(* CoDeSys 2.3.9.50 project: Acp_Bag_2Wrapping_Code.pro *)
(* Libraries: COMlibV2.lib 24.2.14 07:15:46, SysLibAlarmTrend.lib 17.10.05 06:42:38, TcBase.lib 14.5.09 05:44:08, TcSystem.lib 7.6.16 04:31:22, TcUtilities.lib 3.2.16 09:38:58, STANDARD.LIB 5.6.98 05:33:02, TcEtherCAT.lib 30.11.16 13:22:18, SysLibTargetVisu.lib 16.6.08 09:54:26, TcBaseMath.lib 27.7.04 05:37:56, SysLibVisu.lib 7.7.04 11:47:22, TcSystemCX.lib 7.9.16 06:21:26, FB_DateTime.lib 15.2.16 11:06:26, TcMath.lib 23.9.04 08:45:30 *)

(* Task configuration *)
TASK Standard (PRIORITY := 0, INTERVAL := T#10ms);
	MAIN
END_TASK
TASK VISU_TASK (PRIORITY := 3, INTERVAL := T#200ms);
	MAINTARGETVISU_PAINT_CODE
END_TASK
TASK VISU_INPUT_TASK (PRIORITY := 2, INTERVAL := T#50ms);
	MAINTARGETVISU_INPUT_CODE
END_TASK

(* Global variable list: Alarms *)
VAR_GLOBAL
	bAError1: BOOL;
	bAError2: BOOL;
	bAError3: BOOL;
	bAError4: BOOL;
	bAError5: BOOL;
	bAError6: BOOL;
	bAError7: BOOL;
	bAError8: BOOL;
	bAError9: BOOL;
	bAError10: BOOL;
	bAError11: BOOL;
	bAError12: BOOL;
	bAError13: BOOL;
	bAError14: BOOL;
	bAError15: BOOL;
	bAError16: BOOL;
	bAError17: BOOL;
	bAError18: BOOL;
	bAError19: BOOL;
	bAError20: BOOL;
	bAError1Status: STRING;
	bAError2Status: STRING;
	bAError3Status: STRING;
	bAError4Status: STRING;
	bAError5Status: STRING;
	bAError6Status: STRING;
	bAError7Status: STRING;
	bAError8Status: STRING;
	bAError9Status: STRING;
	bAError10Status: STRING;
	bAError11Status: STRING;
	bAError12Status: STRING;
	bAError13Status: STRING;
	bAError14Status: STRING;
	bAError15Status: STRING;
	bAError16Status: STRING;
	bAError17Status: STRING;
	bAError18Status: STRING;
	bAError19Status: STRING;
	bAError20Status: STRING;
END_VAR

(* Global variable list: Auto *)
VAR_GLOBAL
	bQAFeedingConveyorMotor: BOOL;
	bAConeFeedConveyorStart: BOOL;
	bAConeFeedConWait: BOOL;
	bRConePresentInConeFeedCon: BOOL;

	bAConeFeedingPistonHomeRsError: BOOL;
	bQAConeFeedPisOn: BOOL;

	bASealConRdy: BOOL;
	bQAForwardPistonOn: BOOL;
	bQAReversePistonOn: BOOL;

	bAConeTiltingRdy: BOOL;
	ConeFeedPistonRdy: BOOL;
	bAConeFeedCount: BOOL;
	bAConeFeedPisOn: BOOL;
	bAConeFeedingPistonEndRsError: BOOL;
	Cone1Reached: BOOL;
	bAConeFeededCount: INT;
	Cone2Reached: BOOL;
	TotalNoOfCones: INT;

	bAConeFwdRevRdy: BOOL;
	bATiltingPistonOn: BOOL;
	bAConeTiltingPistonEndRsError: BOOL;
	bAFwdRevPisRdy: BOOL;
	bAFwdRevCom: BOOL;
	bAConeTiltingPistonHomeRsError: BOOL;
	bATiltingCylCom: BOOL;
	bAConeTiltingCount: INT;

	bAWrapRdy: BOOL;
	bAForwardPistonOn: BOOL;
	bAReversePistonOn: BOOL;
	bAForwardPisEndRsError: BOOL;
	bAReversePisEndRsError: BOOL;
	bAFwdRevCount: INT;
	bAForwardPisHomeRsError: BOOL;
	bAReversePisHomeRsError: BOOL;
	bAWrappingConRdy: BOOL;

	bAWrapConRdy: BOOL;
	bAWrappingConOn: BOOL;
	bAWrapConeAlaignError: BOOL;
	bAWrapConeAlaignError1: BOOL;
	bAWrappingPisRdy: BOOL;
	bAWrapPiston1On: BOOL;
	bAWrapPiston2On: BOOL;
	bASealingConRdy: BOOL;
	bASheetFeedError: BOOL;
	bAWrapPis1EndRsError: BOOL;
	bAWrapPis2EndRsError: BOOL;
	bAWrappingPisCylCom: BOOL;
	bAWrappingPisCylComInt: BOOL;
	bASealUnitStart: BOOL;


	iBagRowCounter_243: INT;
	bQAColumnStopperPiston: BOOL;
	bABagOperationStarted_243: BOOL;
	bABagUnitRdy_243: BOOL;
	bABagOperationRdy_243: BOOL;
	bQAConePusher2Piston: BOOL;
	bQAColumnReversePiston: BOOL;
	bQAConePusher1Piston: BOOL;
	bABagHalfOpCom_243: BOOL;
	bABagOperationStarted: BOOL;
	bABagOperationComplete: BOOL;
	bQABagHolder: BOOL;
	bQASeparatorplatePiston: BOOL;
	bQABagUp_Down50piston: BOOL;
	bABagOperationComplete_243: BOOL;
	bQABagPusherForwardPiston: BOOL;
	bQABagPusherReversePiston: BOOL;
	TON_bagPusher_243: TON;
	BagOpCom_243: BOOL;
	bForceBagHolder: BOOL;
	bABagComplete: BOOL;
	bQABagTiltingpistonReverse: BOOL;
	bABagTiltingRevOk_243: BOOL;
	bQAColumnConeReversePiston: BOOL;
	bQABagUp_Down180piston: BOOL;
	bQABagTiltingpistonForward: BOOL;
	bQABagBagUp_Down50piston: BOOL;
	bQABagRowHolderpiston: BOOL;

	bASealingConRdy_Bag: BOOL;
	bASealingConRdy_Box: BOOL;
	bASealingUnitOperationCom: BOOL;
	bABoxUnitRdy: BOOL;
	bABoxOperationCom: BOOL;
	bQASealingConFwd1: BOOL;
	bQASealingConRev: BOOL;
	bASealConeSet1Started: BOOL;
	bQASealingConFwd2: BOOL;
	bASealingConeCountEnable: BOOL;
	bASealConeSet1Completed: BOOL;
	bASealConeSet2Started: BOOL;
	bASealConeSet2Completed: BOOL;
	bASealConeRevSetCompleted: BOOL;
	bASealConeMissError: BOOL;
	bASealConeMissErrorStatus: STRING;
	bASealConeMissError1: BOOL;
	bASealConeMissError2: BOOL;
	bASealConeMissError3: BOOL;
	bASealingUnitInt: BOOL;
	bQASealingSeparatorYAxisPiston: BOOL;
	bQASealingTopPiston: BOOL;
	bQASealingBottomPiston: BOOL;
	bQASealingSeparatorXAxisPiston: BOOL;
	bAFilmLoaded1: BOOL;
	bAFilmLoaded2: BOOL;
END_VAR

(* Global variable list: DataLog *)
VAR_GLOBAL
	R_TRIG_IndoPrint: R_TRIG;
	FB_FileOpen_Indo: FB_FileOpen;
	FB_FileWrite_Indo: FB_FileWrite;
	FB_FileClose_Indo: FB_FileClose;
	FB_FileDelete_Indo: FB_FileDelete;
	IndoReport: INT;
	ReportHead1_Indo: BOOL;
	ST1_ProductionData: BOOL;
	ReportHead2_Indo: BOOL;
	ReportBot1_Indo: BOOL;
	stStation1_ProductionData: BOOL;
	ReportBot2_Indo: BOOL;
	testbit: BOOL;
	sOldDay: STRING;
	WriteError: INT;
	OpenError: INT;
	ProductionData_IndoPrint2:STRING(255);
	ProductionDataError_IndoPrint2:STRING(255);
	ProductionDataValues_IndoPrint_Com:STRING(255);
	bANewDay: BOOL;
	SerialNoError: DINT;
	ProductionDataValues_IndoPrint: STRING(255);
	ProductionData_IndoPrint: STRING(255);
	ProductionDataError_IndoPrint: STRING(255);
	ProductionData_ReportData1 : ProductionData_ReportData;
	PROCESSCOMPLETE: BOOL;
	ReportSave: BOOL;
	SerialNo AT %Q*: DINT;
END_VAR

(* Global variable list: Initialize *)
VAR_GLOBAL
	Initialize_TapHmi: BOOL;
	bAInitializeSeq: BOOL;
	bAMachineOn: BOOL;
	bASupplyPressureError: BOOL;
	IntAllOver: BOOL;
	bAIntHomeCheckError: BOOL;

	bQRWappingConveyorMotor: BOOL;
	WrappingConIntRunning: BOOL;
	WrapConIntOver: BOOL;
	bRConePresentInWrapCon: BOOL;
	bQRWrappingPiston1: BOOL;
	bQRWrappingPiston2: BOOL;
	bAWrappingPiston1RsError: BOOL;
	bAWrappingPiston2RsError: BOOL;
	WrapUnitIntOver: BOOL;
	sWrappingConStatus: STRING;
	TiltIntRdy: BOOL;

	bQRForwardPiston: BOOL;
	bQRReversePiston: BOOL;
	bQRTiltingPiston: BOOL;
	bQATiltingPiston: BOOL;
	TiltingIntOvr: BOOL;

	bQRSealingConveyorMotor: BOOL;
	bRConePresentInSealCon: BOOL;
	SealingConIntRunning: BOOL;
	sSealingConStatus: STRING;
	SealConIntOver: BOOL;
	bQRSealingTopPiston: BOOL;
	bQRSealingBottomPiston: BOOL;
	bQRSealingSeparatorXAxisPiston: BOOL;
	bRSealUnitIntOver: BOOL;
	bQRSealingSeparatorYAxisPiston: BOOL;

	bRBagUnitIntRdy: BOOL;
END_VAR

(* Global variable list: Inputs *)
VAR_GLOBAL
					(*I1-EL1809*)

	(*IR1*)	bIUnit_A_RowStopperHome AT %I* : BOOL;
	(*IR2*)	bIUnit_A_RowStopperMiddle AT %I* :BOOL;
	(*IR3*)	bIUnit_A_RowStopperEnd AT %I* :BOOL;
	(*IR4*)	bIUnit_B_RowStopperHome AT %I* :BOOL;
	(*IR5*)	bIUnit_B_RowStopperMiddle AT %I* :BOOL;
	(*IR6*)	bIUnit_B_RowStopperEnd AT %I* :BOOL;
	(*IR7*)	bIUnit_A_ConeDetectionSensor1 AT %I* :BOOL;
	(*IR8*)	bIUnit_A_ConeDetectionSensor2 AT %I* :BOOL;
	(*IR9*)	bIUnit_A_ConeDetectionSensor3 AT %I* :BOOL;
	(*IR10*)	bIUnit_A_ConeDetectionSensor4 AT %I* :BOOL;
	(*IR11*)	bIUnit_A_ConeCrossLimitSwitch AT %I* :BOOL;
	(*IR12*)	bIUnit_B_ConeDetectionSensor1 AT %I* :BOOL;
	(*IR13*)	bIUnit_B_ConeDetectionSensor2 AT %I* :BOOL;
	(*IR14*)	bIUnit_B_ConeDetectionSensor3 AT %I* :BOOL;
	(*IR15*)	bIUnit_B_ConeDetectionSensor4 AT %I* :BOOL;
	(*IR16*)	bIUnit_B_ConeCrossLimitSwitch AT %I* :BOOL;


					(*I2-EL1809*)

	(*IR17*)	bIUnit_AStartPb AT %I* :BOOL;
	(*IR18*)	bIUnit_BStartPb AT %I* :BOOL;
	(*IR19*)	bISpare1 AT %I* :BOOL;
	(*IW1*)	bIMcStartPb AT %I* :BOOL;
	(*IW2*)	bIMcStopPb AT %I* :BOOL;
	(*IW3*)	bIAutoManualSwitch AT %I* :BOOL;
	(*IW4*)	bIEmergencySwitchPb AT %I* :BOOL;
	(*IW5*)	bIProgramKeySwitch AT %I* :BOOL;
	(*IW6*)	bIConeOrientationTopLimitSwitch AT %I* :BOOL;
	(*IW7*)	bIFeedconeStopSensor AT %I* :BOOL;
	(*IW8*)	bIConeFeedingPistonHome AT%I* :BOOL;
	(*IW9*)	bIConeFeedingPistonEnd AT %I* :BOOL;
	(*IW10*)	bIForwardPistonHome AT %I* :BOOL;
	(*IW11*)	bIForwardPistonEnd AT %I* :BOOL;
	(*IW12*)	bIReversePistonHome AT %I* :BOOL;
	(*IW13*)	bIReversePistonEnd AT %I* :BOOL;

						(*I3-EL1809*)

	(*IW14*)	bITiltingHome AT %I* :BOOL;
	(*IW15*)	bITiltingMiddle AT %I* :BOOL;
	(*IW16*)	bITiltingEnd AT %I* :BOOL;
	(*IW17*)	bIWrappingChanelPiston1Home AT %I* :BOOL;
	(*IW18*)	bIWrappingChanelPiston1Middle AT %I* :BOOL;
	(*IW19*)	bIWrappingChanelPiston1End AT %I* :BOOL;
	(*IW20*)	bIWrappingChanelPiston2Home AT %I* :BOOL;
	(*IW21*)	bIWrappingChanelPiston2Middle AT %I* :BOOL;
	(*IW22*)	bIWrappingChanelPiston2End AT %I* :BOOL;
	(*IW23*)	bIWrappingCone1 AT %I* :BOOL;
	(*IW24*)	bIWrappingCone2 AT %I* :BOOL;
	(*IW25*)	bIFilmTensionRod1Home AT %I* :BOOL;
	(*IW26*)	bIFilmTensionRod1End AT %I* :BOOL;
	(*IW27*)	bIFilmTensionRod2Home AT %I* :BOOL;
	(*IW28*)	bIFilmTensionRod2End AT %I* :BOOL;
	(*IW29*)	bISpare2 AT %I* :BOOL;

						(*I4-EL1809*)

	(*IW30*)	bISealingSeparatorYAxisPistonHome AT %I* :BOOL;
	(*IW31*)	bISealingSeparatorYAxisPistoEnd AT %I* :BOOL;
	(*IW32*)	bISealingTopPistonHome AT %I* :BOOL;
	(*IW33*)	bISealingTopPistonEnd AT %I* :BOOL;
	(*IW34*)	bISealingBottomPistonHome AT %I* :BOOL;
	(*IW35*)	bISealingBottomPistonEnd AT %I* :BOOL;
	(*IW36*)	bISealingSeparatorXAxisPistonHome AT %I* :BOOL;
	(*IW37*)	bISealingSeparatorXAxisPistonEnd AT %I* :BOOL;
	(*IW38*)	bIManualSealingPb AT %I* :BOOL;
	(*IW39*)	bIConeCountsensor AT %I* :BOOL;
	(*IW40*)	bIPressureSwitch AT %I* :BOOL;
	(*IW41*)	bIResetPb AT %I* :BOOL;
	(*IW42*)	bIPausePb AT %I* :BOOL;
	(*IW43*)	bIConeCountSensorRev AT %I* :BOOL;
	(*IW44*)	bIConecountStopperPistonHome AT %I* :BOOL;
	(*IW45*)	bIConecountStopperPistonEnd AT%I* :BOOL;


						(*I5-EL1809*)

	(*IW46*)	bIResetSealingPb AT %I* :BOOL;
	(*IW47*)	bISpare4 AT %I* :BOOL;
	(*IW48*)	bISpare5 AT %I* :BOOL;
	(*IW49*)	bISpare6 AT %I* :BOOL;
	(*IW50*)	bISpare7 AT %I* :BOOL;
	(*IW51*)	bISpare8 AT %I* :BOOL;
	(*IW52*)	bISpare9 AT %I* :BOOL;
	(*IW53*)	bISpare10 AT %I*: BOOL;

					(*I6-EL1809*)

	(*IB1*)	bIColumnStopperPistonHome AT %I*: BOOL;
	(*IB2*)	bIColumnStopperPistonEnd AT %I*: BOOL;
	(*IB3*)	bIColumnReversePistonHome AT %I*: BOOL;
	(*IB4*)	bIColumnReversePistonEnd AT %I*: BOOL;
	(*IB5*)	bISeperatorPlatePistonHome AT %I*: BOOL;
	(*IB6*)	bISeperatorPlatePistonEnd AT %I*: BOOL;
	(*IB7*)	bIConePusher1PistonHome AT %I*: BOOL;
	(*IB8*)	bIConePusher1PistonEnd AT %I*: BOOL;
	(*IB9*)	bIConePusher1SaftyObjectSensor AT %I*: BOOL;
	(*IB10*)	bIBagUpDown180PistonHome AT %I*: BOOL;
	(*IB11*)	bIBagUpDown180PistonEnd AT %I*: BOOL;
	(*IB12*)	bIBagUpDown50PistonHome AT %I*: BOOL;
	(*IB13*)	bIBagUpDown50PistonEnd AT %I*: BOOL;
	(*IB14*)	bIBagPusherPistonHome AT %I*: BOOL;
	(*IB15*)	bIBagPusherPistonMiddle AT %I*: BOOL;
	(*IB16*)	bIBagPusherPistonEnd AT %I*: BOOL;

						(*I7-EL1809*)

	(*IB17*)	bIBagTiltingPistonHome AT %I*: BOOL;
	(*IB18*)	bIBagiltingPistonEnd AT %I*: BOOL;
	(*IB19*)	bIBagEmptyCheckObjectSensor AT %I*: BOOL;
	(*IB20*)	bIBagHolderOn  AT %I*: BOOL;
	(*IB21*)	bIBagResetPb AT %I*: BOOL;
	(*IB22*) 	bISpare11 AT %I*: BOOL;
	(*IB23*) 	bISpare12 AT %I*: BOOL;
	(*IB24*) 	bISpare13 AT %I*: BOOL;
END_VAR

(* Global variable list: Main *)
VAR_GLOBAL
	(****************START / STOP / PAUSE / RESUME***************)
	Start_TapHmi: BOOL;
	bAutoModeOn: BOOL;
	bMcStartInAuto: BOOL;
	bMcStopEnable: BOOL;
	Stop_TapHmi: BOOL;
	Pause_TapHmi: BOOL;
	bPauseSeq: BOOL;
	Resume_TapHmi: BOOL;
	Reset_TapHmi: BOOL;
	bErrorReset: BOOL;
	bMcStopEnable1: BOOL;
(*============== Auto/Manual Mode Selection Logic========================*)
	bManualModeOn: BOOL;
	bManualmode: BOOL;
	sMcStatus: STRING;
	bHidePopUp: BOOL;
	bManualModeOk_TapHmi: BOOL;
	bManualModeNOk_TapHmi: BOOL;
(*====================Logic for Model Selection===============*)
	BagSelect_TapHmi: BOOL;
	bAMainIntStarted: BOOL;
	bABoxModeSelected: BOOL;
	BoxSelect_TapHmi: BOOL;
	bABagModeSelected: BOOL;
	sPackingModeStatus: STRING;

	(****************DATE AND TIME***********)
	FB_DateTime_1: FB_DateTime;
	sHourPreFix: STRING;
	sHou: STRING;
	sDayPreFix: STRING;
	sDay: STRING;
	sMonthPreFix: STRING;
	sMonth: STRING;
	sDayF: STRING;
	sMonthF: STRING;
	sDayMonth: STRING;
	sDayF1: STRING;
	sMonthF1: STRING;
	sDayMonth1: STRING;
	sDayMonthYear: STRING;
	sDayMonthYear1: STRING;
	sDaateReport: STRING;
	ReportPath: STRING;
	ReportPath_Final: STRING;
	ReportPath_Final_1: STRING;
	ReportPath_Final_2: STRING;
	sDateReport: STRING;
	ReportPathError: STRING;
	ReportPath_FinalError: STRING;
	ReportPath_Final_1Error: STRING;
	ReportPath_Final_2Error: STRING;
	DateTimeVar: STRING;
	wTodayToHmiFinal: STRING;
(*===============Shift Calculation============*)
	bAShift1Hour: BOOL;
	bAShift2Hour: BOOL;
	bAShift3Hour: BOOL;
	Sfiht1From_Hmi  AT %Q*: WORD;
	Sfiht2From_Hmi  AT %Q*: WORD;
	Sfiht3From_Hmi  AT %Q*: WORD;
	Sfiht1To_Hmi AT %Q*: WORD;
	Sfiht2To_Hmi AT %Q*: WORD;
	Sfiht3To_Hmi AT %Q*: WORD;
	sShitStatus: STRING;
END_VAR

(* Global variable list: Manual *)
VAR_GLOBAL
	WrappingSafety: BOOL;
	SealingSafety: BOOL;
	bManualSealEnable: BOOL;
	bManualSealEnable2: BOOL;
	bMManualSealOn: BOOL;
	bQM_Cone_Sealing_Bottom_Piston: BOOL;
	bQM_Cone_Sealing_Top_Piston: BOOL;
	bHMI_Cone_Forward_Piston_On: BOOL;
	bQM_Cone_Forward_Piston: BOOL;
	bHMI_Cone_Feeding_Piston_On: BOOL;
	bQM_Cone_Feeding_Piston: BOOL;
	bHMI_Cone_Reverse_Piston_On: BOOL;
	bQM_Cone_Reverse_Piston: BOOL;
	bHMI_Cone_Tilting_Piston_On: BOOL;
	bQM_Cone_Tilting_Piston: BOOL;
	bQM_Cone_Tilting_Piston_Rev: BOOL;
	bHMI_Cone_Tilting_Piston_On_Rev: BOOL;
	bHMI_Cone_Wrapping_Piston_On: BOOL;
	bQM_Cone_Wrapping_Piston_Rev: BOOL;
	bQM_Cone_Wrapping_Piston_Fwd: BOOL;
	bHMI_Cone_Wrapping_Piston_On_Rev: BOOL;
	bHMI_Cone_Sealing_Top_Piston_On: BOOL;
	bHMI_Cone_Sealing_Bottom_Piston_On: BOOL;
	bHMI_Cone_Sealing_YAxis_Piston_On: BOOL;
	bQM_Cone_Sealing_YAxis_Piston: BOOL;
	bHMI_Cone_Sealing_XAxis_Piston_On: BOOL;
	bQM_Cone_Sealing_XAxis_Piston: BOOL;
	bHMI_Cone_Feeding_Conveyor_On: BOOL;
	bQM_Cone_Feeding_Conveyor: BOOL;
	bHMI_Cone_Wrapping_Conveyor_On: BOOL;
	bQM_Cone_Wrapping_Conveyor: BOOL;
	bHMI_Cone_Sealing_Conveyor_On: BOOL;
	bQM_Cone_Sealing_Conveyor: BOOL;
	bIConePusher1_On_Hmi: BOOL;
	bQMConePusher1: BOOL;
	bIConePusher2_On_Hmi: BOOL;
	bQMConePusher2: BOOL;
	bIConePusher3_On_Hmi: BOOL;
	bQMConePusher3: BOOL;
	bIBagPusherFwd_On_Hmi: BOOL;
	bQMBagPusherFwd: BOOL;
	bIBagPusherRev_On_Hmi: BOOL;
	bQMBagPusherRev: BOOL;
	bIUpDownPiston_1_On_Hmi: BOOL;
	bQMUpDownPiston_1: BOOL;
	bIUpDownPiston_2_On_Hmi: BOOL;
	bQMUpDownPiston_2: BOOL;
	bIBagTiltingFwd_On_Hmi: BOOL;
	bQMBagTiltingFwd: BOOL;
	bIBagTiltingRev_On_Hmi: BOOL;
	bQMBagTiltingRev: BOOL;
	bIColumn_Stopper_Piston_On_Hmi: BOOL;
	bQMColumnStopperPiston: BOOL;
	bIColumnConeForwardPiston_On_Hmi: BOOL;
	bQMColumnConeForwardPiston: BOOL;
	bIBagHolder_On: BOOL;
	bIBagHolder_On_Hmi: BOOL;
	bIBagPusherHome: BOOL;
	bQMBagHolderPiston: BOOL;
	bHMI_RetA_Fwd_On: BOOL;
	bHMI_RetA_Rev_On: BOOL;
	bQM_RetA_Rev: BOOL;
	bQM_RetA_Fwd: BOOL;
	bHMI_Ret_RevA_On: BOOL;

	bHMI_RetB_Fwd_On: BOOL;
	bHMI_RetB_Rev_On: BOOL;
	bQM_RetB_Rev: BOOL;
	bQM_RetB_Fwd: BOOL;
	bHMI_Ret_RevB_On: BOOL;
	bHMI_Cone_Wrapping_Piston1_On: BOOL;
	bQM_Cone_Wrapping_Piston1_Fwd: BOOL;
	bHMI_Cone_Wrapping_Piston1_On_Rev: BOOL;
	bQM_Cone_Wrapping_Piston1_Rev: BOOL;
	bHMI_Cone_Wrapping_Piston2_On: BOOL;
	bQM_Cone_Wrapping_Piston2_Rev: BOOL;
	bQM_Cone_Wrapping_Piston2_Fwd: BOOL;
	bHMI_Cone_Wrapping_Piston2_On_Rev: BOOL;
	bHMI_Cone_Count_Piston_On: BOOL;
	bQM_Cone_Count_Piston: BOOL;
	bIBagRowHolderPiston_On_Hmi: BOOL;
	bQMBagRowHolderPiston: BOOL;
END_VAR

(* Global variable list: Output_Flags *)
VAR_GLOBAL
	bQAFilmRollerMotor1OnAuto:BOOL;
	bQAFilmRollerMotor2OnAuto: BOOL;
	bQRColumnStopperPiston: BOOL;
	bQMColumnReversePiston: BOOL;
	bQMSeparatorplatePiston: BOOL;
	bQMConePusher1Piston: BOOL;
	bQMConePusher2Piston: BOOL;
	bQMBagPusherForwardPiston: BOOL;
	bQMBagPusherReversePiston: BOOL;
	bQMBagUp_Down180piston: BOOL;
	bQMBagUp_Down50piston: BOOL;
	bQMBagTiltingpistonForward: BOOL;
	bQMBagTiltingpistonReverse: BOOL;
	bQMSpareOutput13: BOOL;
	bQMSpareOutput14: BOOL;
	bQMSpareOutput15: BOOL;
	bQRColumnReversePiston: BOOL;
	bQRSeparatorplatePiston: BOOL;
	bQRConePusher1Piston: BOOL;
	bQRConePusher2Piston: BOOL;
	bQRBagPusherForwardPiston: BOOL;
	bQRBagPusherReversePiston: BOOL;
	bQRBagHolderpiston: BOOL;
	bQRBagUp_Down180piston: BOOL;
	bQRBagUp_Down50piston: BOOL;
	bQRBagTiltingpistonForward: BOOL;
	bQRBagTiltingpistonReverse: BOOL;
	bQRSpareOutput13: BOOL;
	bQRSpareOutput14: BOOL;
	bQRSpareOutput15: BOOL;
	bAQColumnReversePiston: BOOL;
	bQABagHolderpiston: BOOL;
	bQASpareOutput13: BOOL;
	bQASpareOutput14: BOOL;
	bQASpareOutput15: BOOL;
	bQMSpareOutput5: BOOL;
	bQRSpareOutput5: BOOL;
	bQASpareOutput5: BOOL;
	bQMSpareOutput6: BOOL;
	bQRSpareOutput6: BOOL;
	bQASpareOutput6: BOOL;
	bQMSpareOutput7: BOOL;
	bQRSpareOutput7: BOOL;
	bQASpareOutput7: BOOL;
	bQMSpareOutput8: BOOL;
	bQRSpareOutput8: BOOL;
	bQASpareOutput8: BOOL;
	bQMSpareOutput9: BOOL;
	bQRSpareOutput9: BOOL;
	bQASpareOutput9: BOOL;
	bQMSpareOutput10: BOOL;
	bQRSpareOutput10: BOOL;
	bQASpareOutput10: BOOL;
	bQMSpareOutput11: BOOL;
	bQRSpareOutput11: BOOL;
	bQASpareOutput11: BOOL;
	bQMSpareOutput12: BOOL;
	bQRSpareOutput12: BOOL;
	bQASpareOutput12: BOOL;
	bQMConeFeedingPiston: BOOL;
	bQRConeFeedingPiston: BOOL;
	bQMForwardPiston: BOOL;
	bQMReversePiston: BOOL;
	bQMTiltingPiston: BOOL;
	bQMWrappingPiston1: BOOL;
	bQMWrappingPiston2: BOOL;
	bQMSealingSeparatorYAxisPiston: BOOL;
	bQMSealingTopPiston: BOOL;
	bQMSealingBottomPiston: BOOL;
	bQMSealingSeparatorXAxisPiston: BOOL;
	bQMFilmRollerMotor1: BOOL;
	bQAFilmRollerMotor1: BOOL;
	bQMFilmRollerMotor2: BOOL;
	bQAFilmRollerMotor2: BOOL;
	bQMConeCountPiston: BOOL;
	bQAConeCountPiston: BOOL;
	bQMFeedingConveyorMotor: BOOL;
	bQMWappingConveyorMotor: BOOL;
	bQAWappingConveyorMotor: BOOL;
	bQMSealingConveyorMotor: BOOL;
	bQASealingConveyorMotor: BOOL;
	bQMRetA_RowStopperMotorFwd: BOOL;
	bQRRetA_RowStopperMotorFwd: BOOL;
	bQMRetA_RowStopperMotorRev: BOOL;
	bQRRetA_RowStopperMotorRev: BOOL;
	bQMRetB_RowStopperMotorFwd: BOOL;
	bQRRetB_RowStopperMotorFwd: BOOL;
	bQMRetB_RowStopperMotorRev: BOOL;
	bQRRetB_RowStopperMotorRev: BOOL;
	bQMSpareOutput1: BOOL;
	bQRSpareOutput1: BOOL;
	bQARetA_WeightOk: BOOL;
	bQARetA_WeightNOk: BOOL;
	bQARetB_WeightOk: BOOL;
	bQARetB_WeightNOk: BOOL;
	bQMSpareOutput2: BOOL;
	bQRSpareOutput2: BOOL;
	bQMSpareOutput3: BOOL;
	bQRSpareOutput3: BOOL;
	bQMSpareOutput4: BOOL;
	bQRSpareOutput4: BOOL;
	bQMTowerLampRed: BOOL;
	bQRTowerLampRed: BOOL;
	bQMTowerLampGreen: BOOL;
	bQRTowerLampGreen: BOOL;
	bQMTowerLampYellow: BOOL;
	bQRTowerLampYellow: BOOL;
	bQMTowerBuzzer: BOOL;
	bQRTowerBuzzer: BOOL;
	bQARetA_RowStopperMotorFwd: BOOL;
	bQARetA_RowStopperMotorRev: BOOL;
	bQARetB_RowStopperMotorFwd: BOOL;
	bQARetB_RowStopperMotorRev: BOOL;
	bQASpareOutput1: BOOL;
	bQASpareOutput2: BOOL;
	bQASpareOutput3: BOOL;
	bQASpareOutput4: BOOL;
	bQATowerLampRed: BOOL;
	bQATowerLampGreen: BOOL;
	bQATowerLampYellow: BOOL;
	bQATowerBuzzer: BOOL;
	bQAForwardPiston: BOOL;
	bQAReversePiston: BOOL;
	bQAWrappingPiston1: BOOL;
	bQAWrappingPiston2: BOOL;
	bQRConeCountPiston: BOOL;
	bQRFeedingConveyorMotor: BOOL;

	bQBagHolder: BOOL;
	bQAConePusher3Piston: BOOL;
	bAConePusher1SafetyError: BOOL;
	bAConePusher1SafetyErrorStatus: STRING;

END_VAR

(* Global variable list: Outputs *)
VAR_GLOBAL
				(*O1-EL2809*)

	bQRetA_RowStopperMotorFwd AT %Q* :BOOL;(*OR1*)
	bQRetA_RowStopperMotorRev AT %Q* :BOOL;(*OR2*)
	bQRetB_RowStopperMotorFwd AT %Q* :BOOL;(*OR3*)
	bQRetB_RowStopperMotorRev AT %Q* :BOOL;(*OR4*)
	bQSpareOutput1 AT %Q* :BOOL;(*OR5*)
	bQRetA_WeightOk AT %Q* :BOOL;(*OR6*)
	bQRetA_WeightNOk AT %Q* :BOOL;(*OR7*)
	bQRetB_WeightOk AT %Q* :BOOL;(*OR8*)
	bQRetB_WeightNOk AT %Q* :BOOL;(*OR9*)
	bQSpareOutput2 AT %Q* :BOOL;(*OR10*)
	bQSpareOutput3 AT %Q* :BOOL;(*OR11*)
	bQSpareOutput4 AT %Q* :BOOL;(*OR12*)
	bQTowerLampRed AT %Q* :BOOL;(*R1*)
	bQTowerLampGreen AT %Q* :BOOL;(*R2*)
	bQTowerLampYellow AT %Q* :BOOL;(*R3*)
	bQTowerBuzzer AT %Q* :BOOL;(*R4*)


			(*O2-EL2809*)

	bQConeFeedingPiston AT %Q* :BOOL;(*OW1*)
	bQForwardPiston AT %Q* :BOOL;(*OW2*)
	bQReversePiston AT %Q* :BOOL;(*OW3*)
	bQTiltingPiston AT %Q* :BOOL;(*OW4*)
	bQWrappingPiston1 AT %Q* :BOOL;(*OW5*)
	bQWrappingPiston2 AT %Q* :BOOL;(*OW6*)
	bQSealingSeparatorYAxisPiston AT %Q* :BOOL;(*OW7*)
	bQSealingTopPiston AT %Q* :BOOL;(*OW8*)
	bQSealingBottomPiston AT %Q* :BOOL;(*OW9*)
	bQSealingSeparatorXAxisPiston AT %Q* :BOOL;(*OW10*)
	bQFilmRollerMotor1 AT %Q* :BOOL;(*OW11*)
	bQFilmRollerMotor2 AT %Q* :BOOL;(*OW12*)
	bQConeCountPiston AT %Q* :BOOL;(*OW13*)
	bQFeedingConveyorMotor AT %Q* :BOOL;(*OW14*)
	bQWappingConveyorMotor AT %Q* :BOOL;(*OW15*)
	bQSealingConveyorMotor AT %Q* :BOOL;(*OW16*)



			(*O3-EL2008*)

	bQSpareOutput5 AT %Q* :BOOL;(*OW20*)
	bQSpareOutput6 AT %Q* :BOOL;(*OW21*)
	bQSpareOutput7 AT %Q* :BOOL;(*OW22*)
	bQSpareOutput8 AT %Q* :BOOL;(*OW23*)
	bQSpareOutput9 AT %Q* :BOOL;(*OW24*)
	bQSpareOutput10 AT %Q* :BOOL;(*OW25*)
	bQSpareOutput11 AT %Q* :BOOL;(*OW26*)
	bQSpareOutput12 AT %Q* :BOOL;(*OW27*)

			(*O4-EL2809*)

	bQColumnStopperPiston AT %Q* :BOOL;(*OB1*)
	bQColumnReversePiston AT %Q* :BOOL;(*OB2*)
	bQSeparatorplatePiston AT %Q* :BOOL;(*OB3*)
	bQConePusher1Piston AT %Q* :BOOL;(*OB4*)
	bQConePusher2Piston AT %Q* :BOOL;(*OB5*)
	bQBagPusherForwardPiston AT %Q* :BOOL;(*OB6*)
	bQBagPusherReversePiston AT %Q* :BOOL;(*OB7*)
	bQBagHolderpiston AT %Q* :BOOL;(*OB8*)
	bQBagUp_Down180piston AT %Q* :BOOL;(*OB9*)
	bQBagUp_Down50piston AT %Q* :BOOL;(*OB10*)
	bQBagTiltingpistonForward AT %Q* :BOOL;(*OB11*)
	bQBagTiltingpistonReverse AT %Q* :BOOL;(*OB12*)
	bQBagRowHolderpiston AT %Q* :BOOL;(*OB13*)
	bQSpareOutput13 AT %Q* :BOOL;(*OB14*)
	bQSpareOutput14 AT %Q* :BOOL;(*OB15*)
	bQSpareOutput15 AT %Q* :BOOL;(*OB16*)

END_VAR

(* Global variable list: Parameters *)
VAR_GLOBAL
	Default_NetWeight_Report: STRING;
	Default_GrossWeight_Report: STRING;
	Actual_NetWeight_Report: STRING;
	Actual_GrossWeight_Report: STRING;
	COUNT_DIS: STRING;
	BLEND_DIS: STRING;
	LOTNO_DIS: STRING;
	CARTONNO_DIS: DINT;
	SHADE_DIS: STRING;
END_VAR

(* Global variable list: Print *)
VAR_GLOBAL
	PrintEnabled: BOOL;
	PrintValue: INT;
	PrintEnable_TogHmi: BOOL;
	ProductionData_PrintData: ProductionData_PrintData;
	ProductionDataValues_Print: STRING(255);
	ProductionDataValues_Print_Com:STRING(255);
	ProductionData_Print: STRING(255);
	FB_FileOpen1: FB_FileOpen;
	FB_FileWrite1: FB_FileWrite;
	FB_FileClose1: FB_FileClose;
	FB_FileDelete1: FB_FileDelete;
	PrintOk: BOOL;
END_VAR

(* Global variable list: TwinCAT_Configuration *)
(* Generated automatically by TwinCAT - (read only) *)
VAR_CONFIG
	Weight_Read.COMin_1_COMPort_1 AT %IB0 : EL6inData22B;
	Weight_Read.COMOut_1_COMPort_1 AT %QB0 : EL6outData22B;
	Weight_Read.COMin_2_COMPort_2 AT %IB24 : EL6inData22B;
	Weight_Read.COMOut_2_COMPort_2 AT %QB24 : EL6outData22B;
	.SerialNo AT %QB48 : DINT;
	.bIUnit_A_RowStopperHome AT %IX48.0 : BOOL;	(*  ~ {LinkedWith:TIID^Device 3 (EtherCAT)^Term 1 (EK1100)^Term 2 (EL1809)^Channel 1^Input} *)
	.bIUnit_A_RowStopperMiddle AT %IX48.1 : BOOL;	(*  ~ {LinkedWith:TIID^Device 3 (EtherCAT)^Term 1 (EK1100)^Term 2 (EL1809)^Channel 2^Input} *)
	.bIUnit_A_RowStopperEnd AT %IX48.2 : BOOL;	(*  ~ {LinkedWith:TIID^Device 3 (EtherCAT)^Term 1 (EK1100)^Term 2 (EL1809)^Channel 3^Input} *)
	.bIUnit_B_RowStopperHome AT %IX48.3 : BOOL;	(*  ~ {LinkedWith:TIID^Device 3 (EtherCAT)^Term 1 (EK1100)^Term 2 (EL1809)^Channel 4^Input} *)
	.bIUnit_B_RowStopperMiddle AT %IX48.4 : BOOL;	(*  ~ {LinkedWith:TIID^Device 3 (EtherCAT)^Term 1 (EK1100)^Term 2 (EL1809)^Channel 5^Input} *)
	.bIUnit_B_RowStopperEnd AT %IX48.5 : BOOL;	(*  ~ {LinkedWith:TIID^Device 3 (EtherCAT)^Term 1 (EK1100)^Term 2 (EL1809)^Channel 6^Input} *)
	.bIUnit_A_ConeDetectionSensor1 AT %IX48.6 : BOOL;	(*  ~ {LinkedWith:TIID^Device 3 (EtherCAT)^Term 1 (EK1100)^Term 2 (EL1809)^Channel 7^Input} *)
	.bIUnit_A_ConeDetectionSensor2 AT %IX48.7 : BOOL;	(*  ~ {LinkedWith:TIID^Device 3 (EtherCAT)^Term 1 (EK1100)^Term 2 (EL1809)^Channel 8^Input} *)
	.bIUnit_A_ConeDetectionSensor3 AT %IX49.0 : BOOL;	(*  ~ {LinkedWith:TIID^Device 3 (EtherCAT)^Term 1 (EK1100)^Term 2 (EL1809)^Channel 9^Input} *)
	.bIUnit_A_ConeDetectionSensor4 AT %IX49.1 : BOOL;	(*  ~ {LinkedWith:TIID^Device 3 (EtherCAT)^Term 1 (EK1100)^Term 2 (EL1809)^Channel 10^Input} *)
	.bIUnit_A_ConeCrossLimitSwitch AT %IX49.2 : BOOL;	(*  ~ {LinkedWith:TIID^Device 3 (EtherCAT)^Term 1 (EK1100)^Term 2 (EL1809)^Channel 11^Input} *)
	.bIUnit_B_ConeDetectionSensor1 AT %IX49.3 : BOOL;	(*  ~ {LinkedWith:TIID^Device 3 (EtherCAT)^Term 1 (EK1100)^Term 2 (EL1809)^Channel 12^Input} *)
	.bIUnit_B_ConeDetectionSensor2 AT %IX49.4 : BOOL;	(*  ~ {LinkedWith:TIID^Device 3 (EtherCAT)^Term 1 (EK1100)^Term 2 (EL1809)^Channel 13^Input} *)
	.bIUnit_B_ConeDetectionSensor3 AT %IX49.5 : BOOL;	(*  ~ {LinkedWith:TIID^Device 3 (EtherCAT)^Term 1 (EK1100)^Term 2 (EL1809)^Channel 14^Input} *)
	.bIUnit_B_ConeDetectionSensor4 AT %IX49.6 : BOOL;	(*  ~ {LinkedWith:TIID^Device 3 (EtherCAT)^Term 1 (EK1100)^Term 2 (EL1809)^Channel 15^Input} *)
	.bIUnit_B_ConeCrossLimitSwitch AT %IX49.7 : BOOL;	(*  ~ {LinkedWith:TIID^Device 3 (EtherCAT)^Term 1 (EK1100)^Term 2 (EL1809)^Channel 16^Input} *)
	.bIUnit_AStartPb AT %IX50.0 : BOOL;	(*  ~ {LinkedWith:TIID^Device 3 (EtherCAT)^Term 1 (EK1100)^Term 3 (EL1809)^Channel 1^Input} *)
	.bIUnit_BStartPb AT %IX50.1 : BOOL;	(*  ~ {LinkedWith:TIID^Device 3 (EtherCAT)^Term 1 (EK1100)^Term 3 (EL1809)^Channel 2^Input} *)
	.bISpare1 AT %IX50.2 : BOOL;	(*  ~ {LinkedWith:TIID^Device 3 (EtherCAT)^Term 1 (EK1100)^Term 3 (EL1809)^Channel 3^Input} *)
	.bIMcStartPb AT %IX50.3 : BOOL;	(*  ~ {LinkedWith:TIID^Device 3 (EtherCAT)^Term 1 (EK1100)^Term 3 (EL1809)^Channel 4^Input} *)
	.bIMcStopPb AT %IX50.4 : BOOL;	(*  ~ {LinkedWith:TIID^Device 3 (EtherCAT)^Term 1 (EK1100)^Term 3 (EL1809)^Channel 5^Input} *)
	.bIAutoManualSwitch AT %IX50.5 : BOOL;	(*  ~ {LinkedWith:TIID^Device 3 (EtherCAT)^Term 1 (EK1100)^Term 3 (EL1809)^Channel 6^Input} *)
	.bIEmergencySwitchPb AT %IX50.6 : BOOL;	(*  ~ {LinkedWith:TIID^Device 3 (EtherCAT)^Term 1 (EK1100)^Term 3 (EL1809)^Channel 7^Input} *)
	.bIProgramKeySwitch AT %IX50.7 : BOOL;	(*  ~ {LinkedWith:TIID^Device 3 (EtherCAT)^Term 1 (EK1100)^Term 3 (EL1809)^Channel 8^Input} *)
	.bIConeOrientationTopLimitSwitch AT %IX51.0 : BOOL;	(*  ~ {LinkedWith:TIID^Device 3 (EtherCAT)^Term 1 (EK1100)^Term 3 (EL1809)^Channel 9^Input} *)
	.bIFeedconeStopSensor AT %IX51.1 : BOOL;	(*  ~ {LinkedWith:TIID^Device 3 (EtherCAT)^Term 1 (EK1100)^Term 3 (EL1809)^Channel 10^Input} *)
	.bIConeFeedingPistonHome AT %IX51.2 : BOOL;	(*  ~ {LinkedWith:TIID^Device 3 (EtherCAT)^Term 1 (EK1100)^Term 3 (EL1809)^Channel 11^Input} *)
	.bIConeFeedingPistonEnd AT %IX51.3 : BOOL;	(*  ~ {LinkedWith:TIID^Device 3 (EtherCAT)^Term 1 (EK1100)^Term 3 (EL1809)^Channel 12^Input} *)
	.bIForwardPistonHome AT %IX51.4 : BOOL;	(*  ~ {LinkedWith:TIID^Device 3 (EtherCAT)^Term 1 (EK1100)^Term 3 (EL1809)^Channel 13^Input} *)
	.bIForwardPistonEnd AT %IX51.5 : BOOL;	(*  ~ {LinkedWith:TIID^Device 3 (EtherCAT)^Term 1 (EK1100)^Term 3 (EL1809)^Channel 14^Input} *)
	.bIReversePistonHome AT %IX51.6 : BOOL;	(*  ~ {LinkedWith:TIID^Device 3 (EtherCAT)^Term 1 (EK1100)^Term 3 (EL1809)^Channel 15^Input} *)
	.bIReversePistonEnd AT %IX51.7 : BOOL;	(*  ~ {LinkedWith:TIID^Device 3 (EtherCAT)^Term 1 (EK1100)^Term 3 (EL1809)^Channel 16^Input} *)
	.bITiltingHome AT %IX52.0 : BOOL;	(*  ~ {LinkedWith:TIID^Device 3 (EtherCAT)^Term 1 (EK1100)^Term 4 (EL1809)^Channel 1^Input} *)
	.bITiltingMiddle AT %IX52.1 : BOOL;	(*  ~ {LinkedWith:TIID^Device 3 (EtherCAT)^Term 1 (EK1100)^Term 4 (EL1809)^Channel 2^Input} *)
	.bITiltingEnd AT %IX52.2 : BOOL;	(*  ~ {LinkedWith:TIID^Device 3 (EtherCAT)^Term 1 (EK1100)^Term 4 (EL1809)^Channel 3^Input} *)
	.bIWrappingChanelPiston1Home AT %IX52.3 : BOOL;	(*  ~ {LinkedWith:TIID^Device 3 (EtherCAT)^Term 1 (EK1100)^Term 4 (EL1809)^Channel 4^Input} *)
	.bIWrappingChanelPiston1Middle AT %IX52.4 : BOOL;	(*  ~ {LinkedWith:TIID^Device 3 (EtherCAT)^Term 1 (EK1100)^Term 4 (EL1809)^Channel 5^Input} *)
	.bIWrappingChanelPiston1End AT %IX52.5 : BOOL;	(*  ~ {LinkedWith:TIID^Device 3 (EtherCAT)^Term 1 (EK1100)^Term 4 (EL1809)^Channel 6^Input} *)
	.bIWrappingChanelPiston2Home AT %IX52.6 : BOOL;	(*  ~ {LinkedWith:TIID^Device 3 (EtherCAT)^Term 1 (EK1100)^Term 4 (EL1809)^Channel 7^Input} *)
	.bIWrappingChanelPiston2Middle AT %IX52.7 : BOOL;	(*  ~ {LinkedWith:TIID^Device 3 (EtherCAT)^Term 1 (EK1100)^Term 4 (EL1809)^Channel 8^Input} *)
	.bIWrappingChanelPiston2End AT %IX53.0 : BOOL;	(*  ~ {LinkedWith:TIID^Device 3 (EtherCAT)^Term 1 (EK1100)^Term 4 (EL1809)^Channel 9^Input} *)
	.bIWrappingCone1 AT %IX53.1 : BOOL;	(*  ~ {LinkedWith:TIID^Device 3 (EtherCAT)^Term 1 (EK1100)^Term 4 (EL1809)^Channel 10^Input} *)
	.bIWrappingCone2 AT %IX53.2 : BOOL;	(*  ~ {LinkedWith:TIID^Device 3 (EtherCAT)^Term 1 (EK1100)^Term 4 (EL1809)^Channel 11^Input} *)
	.bIFilmTensionRod1Home AT %IX53.3 : BOOL;	(*  ~ {LinkedWith:TIID^Device 3 (EtherCAT)^Term 1 (EK1100)^Term 4 (EL1809)^Channel 12^Input} *)
	.bIFilmTensionRod1End AT %IX53.4 : BOOL;	(*  ~ {LinkedWith:TIID^Device 3 (EtherCAT)^Term 1 (EK1100)^Term 4 (EL1809)^Channel 13^Input} *)
	.bIFilmTensionRod2Home AT %IX53.5 : BOOL;	(*  ~ {LinkedWith:TIID^Device 3 (EtherCAT)^Term 1 (EK1100)^Term 4 (EL1809)^Channel 14^Input} *)
	.bIFilmTensionRod2End AT %IX53.6 : BOOL;	(*  ~ {LinkedWith:TIID^Device 3 (EtherCAT)^Term 1 (EK1100)^Term 4 (EL1809)^Channel 15^Input} *)
	.bISpare2 AT %IX53.7 : BOOL;	(*  ~ {LinkedWith:TIID^Device 3 (EtherCAT)^Term 1 (EK1100)^Term 4 (EL1809)^Channel 16^Input} *)
	.bISealingSeparatorYAxisPistonHome AT %IX54.0 : BOOL;	(*  ~ {LinkedWith:TIID^Device 3 (EtherCAT)^Term 1 (EK1100)^Term 5 (EL1809)^Channel 1^Input} *)
	.bISealingSeparatorYAxisPistoEnd AT %IX54.1 : BOOL;	(*  ~ {LinkedWith:TIID^Device 3 (EtherCAT)^Term 1 (EK1100)^Term 5 (EL1809)^Channel 2^Input} *)
	.bISealingTopPistonHome AT %IX54.2 : BOOL;	(*  ~ {LinkedWith:TIID^Device 3 (EtherCAT)^Term 1 (EK1100)^Term 5 (EL1809)^Channel 3^Input} *)
	.bISealingTopPistonEnd AT %IX54.3 : BOOL;	(*  ~ {LinkedWith:TIID^Device 3 (EtherCAT)^Term 1 (EK1100)^Term 5 (EL1809)^Channel 4^Input} *)
	.bISealingBottomPistonHome AT %IX54.4 : BOOL;	(*  ~ {LinkedWith:TIID^Device 3 (EtherCAT)^Term 1 (EK1100)^Term 5 (EL1809)^Channel 5^Input} *)
	.bISealingBottomPistonEnd AT %IX54.5 : BOOL;	(*  ~ {LinkedWith:TIID^Device 3 (EtherCAT)^Term 1 (EK1100)^Term 5 (EL1809)^Channel 6^Input} *)
	.bISealingSeparatorXAxisPistonHome AT %IX54.6 : BOOL;	(*  ~ {LinkedWith:TIID^Device 3 (EtherCAT)^Term 1 (EK1100)^Term 5 (EL1809)^Channel 7^Input} *)
	.bISealingSeparatorXAxisPistonEnd AT %IX54.7 : BOOL;	(*  ~ {LinkedWith:TIID^Device 3 (EtherCAT)^Term 1 (EK1100)^Term 5 (EL1809)^Channel 8^Input} *)
	.bIManualSealingPb AT %IX55.0 : BOOL;	(*  ~ {LinkedWith:TIID^Device 3 (EtherCAT)^Term 1 (EK1100)^Term 5 (EL1809)^Channel 9^Input} *)
	.bIConeCountsensor AT %IX55.1 : BOOL;	(*  ~ {LinkedWith:TIID^Device 3 (EtherCAT)^Term 1 (EK1100)^Term 5 (EL1809)^Channel 10^Input} *)
	.bIPressureSwitch AT %IX55.2 : BOOL;	(*  ~ {LinkedWith:TIID^Device 3 (EtherCAT)^Term 1 (EK1100)^Term 5 (EL1809)^Channel 11^Input} *)
	.bIResetPb AT %IX55.3 : BOOL;	(*  ~ {LinkedWith:TIID^Device 3 (EtherCAT)^Term 1 (EK1100)^Term 5 (EL1809)^Channel 12^Input} *)
	.bIPausePb AT %IX55.4 : BOOL;	(*  ~ {LinkedWith:TIID^Device 3 (EtherCAT)^Term 1 (EK1100)^Term 5 (EL1809)^Channel 13^Input} *)
	.bIConeCountSensorRev AT %IX55.5 : BOOL;	(*  ~ {LinkedWith:TIID^Device 3 (EtherCAT)^Term 1 (EK1100)^Term 5 (EL1809)^Channel 14^Input} *)
	.bIConecountStopperPistonHome AT %IX55.6 : BOOL;	(*  ~ {LinkedWith:TIID^Device 3 (EtherCAT)^Term 1 (EK1100)^Term 5 (EL1809)^Channel 15^Input} *)
	.bIConecountStopperPistonEnd AT %IX55.7 : BOOL;	(*  ~ {LinkedWith:TIID^Device 3 (EtherCAT)^Term 1 (EK1100)^Term 5 (EL1809)^Channel 16^Input} *)
	.bIResetSealingPb AT %IX56.0 : BOOL;	(*  ~ {LinkedWith:TIID^Device 3 (EtherCAT)^Term 1 (EK1100)^Term 7 (EL1008)^Channel 6^Input} *)
	.bISpare4 AT %IX56.1 : BOOL;	(*  ~ {LinkedWith:TIID^Device 3 (EtherCAT)^Term 1 (EK1100)^Term 8 (EL1008)^Channel 1^Input} *)
	.bISpare5 AT %IX56.2 : BOOL;	(*  ~ {LinkedWith:TIID^Device 3 (EtherCAT)^Term 1 (EK1100)^Term 8 (EL1008)^Channel 2^Input} *)
	.bISpare6 AT %IX56.3 : BOOL;	(*  ~ {LinkedWith:TIID^Device 3 (EtherCAT)^Term 1 (EK1100)^Term 8 (EL1008)^Channel 3^Input} *)
	.bISpare7 AT %IX56.4 : BOOL;	(*  ~ {LinkedWith:TIID^Device 3 (EtherCAT)^Term 1 (EK1100)^Term 8 (EL1008)^Channel 4^Input} *)
	.bISpare8 AT %IX56.5 : BOOL;	(*  ~ {LinkedWith:TIID^Device 3 (EtherCAT)^Term 1 (EK1100)^Term 8 (EL1008)^Channel 5^Input} *)
	.bISpare9 AT %IX56.6 : BOOL;	(*  ~ {LinkedWith:TIID^Device 3 (EtherCAT)^Term 1 (EK1100)^Term 8 (EL1008)^Channel 6^Input} *)
	.bISpare10 AT %IX56.7 : BOOL;	(*  ~ {LinkedWith:TIID^Device 3 (EtherCAT)^Term 1 (EK1100)^Term 8 (EL1008)^Channel 7^Input} *)
	.bIColumnStopperPistonHome AT %IX57.0 : BOOL;	(*  ~ {LinkedWith:TIID^Device 3 (EtherCAT)^Term 1 (EK1100)^Term 6 (EL1809)^Channel 1^Input} *)
	.bIColumnStopperPistonEnd AT %IX57.1 : BOOL;	(*  ~ {LinkedWith:TIID^Device 3 (EtherCAT)^Term 1 (EK1100)^Term 6 (EL1809)^Channel 2^Input} *)
	.bIColumnReversePistonHome AT %IX57.2 : BOOL;	(*  ~ {LinkedWith:TIID^Device 3 (EtherCAT)^Term 1 (EK1100)^Term 6 (EL1809)^Channel 3^Input} *)
	.bIColumnReversePistonEnd AT %IX57.3 : BOOL;	(*  ~ {LinkedWith:TIID^Device 3 (EtherCAT)^Term 1 (EK1100)^Term 6 (EL1809)^Channel 4^Input} *)
	.bISeperatorPlatePistonHome AT %IX57.4 : BOOL;	(*  ~ {LinkedWith:TIID^Device 3 (EtherCAT)^Term 1 (EK1100)^Term 6 (EL1809)^Channel 5^Input} *)
	.bISeperatorPlatePistonEnd AT %IX57.5 : BOOL;	(*  ~ {LinkedWith:TIID^Device 3 (EtherCAT)^Term 1 (EK1100)^Term 6 (EL1809)^Channel 6^Input} *)
	.bIConePusher1PistonHome AT %IX57.6 : BOOL;	(*  ~ {LinkedWith:TIID^Device 3 (EtherCAT)^Term 1 (EK1100)^Term 6 (EL1809)^Channel 7^Input} *)
	.bIConePusher1PistonEnd AT %IX57.7 : BOOL;	(*  ~ {LinkedWith:TIID^Device 3 (EtherCAT)^Term 1 (EK1100)^Term 6 (EL1809)^Channel 8^Input} *)
	.bIConePusher1SaftyObjectSensor AT %IX58.0 : BOOL;	(*  ~ {LinkedWith:TIID^Device 3 (EtherCAT)^Term 1 (EK1100)^Term 6 (EL1809)^Channel 9^Input} *)
	.bIBagUpDown180PistonHome AT %IX58.1 : BOOL;	(*  ~ {LinkedWith:TIID^Device 3 (EtherCAT)^Term 1 (EK1100)^Term 6 (EL1809)^Channel 10^Input} *)
	.bIBagUpDown180PistonEnd AT %IX58.2 : BOOL;	(*  ~ {LinkedWith:TIID^Device 3 (EtherCAT)^Term 1 (EK1100)^Term 6 (EL1809)^Channel 11^Input} *)
	.bIBagUpDown50PistonHome AT %IX58.3 : BOOL;	(*  ~ {LinkedWith:TIID^Device 3 (EtherCAT)^Term 1 (EK1100)^Term 6 (EL1809)^Channel 12^Input} *)
	.bIBagUpDown50PistonEnd AT %IX58.4 : BOOL;	(*  ~ {LinkedWith:TIID^Device 3 (EtherCAT)^Term 1 (EK1100)^Term 6 (EL1809)^Channel 13^Input} *)
	.bIBagPusherPistonHome AT %IX58.5 : BOOL;	(*  ~ {LinkedWith:TIID^Device 3 (EtherCAT)^Term 1 (EK1100)^Term 6 (EL1809)^Channel 14^Input} *)
	.bIBagPusherPistonMiddle AT %IX58.6 : BOOL;	(*  ~ {LinkedWith:TIID^Device 3 (EtherCAT)^Term 1 (EK1100)^Term 6 (EL1809)^Channel 15^Input} *)
	.bIBagPusherPistonEnd AT %IX58.7 : BOOL;	(*  ~ {LinkedWith:TIID^Device 3 (EtherCAT)^Term 1 (EK1100)^Term 6 (EL1809)^Channel 16^Input} *)
	.bIBagTiltingPistonHome AT %IX59.0 : BOOL;	(*  ~ {LinkedWith:TIID^Device 3 (EtherCAT)^Term 1 (EK1100)^Term 7 (EL1008)^Channel 1^Input} *)
	.bIBagiltingPistonEnd AT %IX59.1 : BOOL;	(*  ~ {LinkedWith:TIID^Device 3 (EtherCAT)^Term 1 (EK1100)^Term 7 (EL1008)^Channel 2^Input} *)
	.bIBagEmptyCheckObjectSensor AT %IX59.2 : BOOL;	(*  ~ {LinkedWith:TIID^Device 3 (EtherCAT)^Term 1 (EK1100)^Term 7 (EL1008)^Channel 3^Input} *)
	.bIBagHolderOn AT %IX59.3 : BOOL;	(*  ~ {LinkedWith:TIID^Device 3 (EtherCAT)^Term 1 (EK1100)^Term 7 (EL1008)^Channel 4^Input} *)
	.bIBagResetPb AT %IX59.4 : BOOL;	(*  ~ {LinkedWith:TIID^Device 3 (EtherCAT)^Term 1 (EK1100)^Term 7 (EL1008)^Channel 5^Input} *)
	.bISpare11 AT %IX59.5 : BOOL;	(*  ~ {LinkedWith:TIID^Device 3 (EtherCAT)^Term 1 (EK1100)^Term 8 (EL1008)^Channel 8^Input} *)
	.bISpare12 AT %IX59.6 : BOOL;	(*  ~ {LinkedWith:TIID^Device 3 (EtherCAT)^Term 1 (EK1100)^Term 7 (EL1008)^Channel 7^Input} *)
	.bISpare13 AT %IX59.7 : BOOL;	(*  ~ {LinkedWith:TIID^Device 3 (EtherCAT)^Term 1 (EK1100)^Term 7 (EL1008)^Channel 8^Input} *)
	.Sfiht1From_Hmi AT %QB52 : WORD;
	.Sfiht2From_Hmi AT %QB54 : WORD;
	.Sfiht3From_Hmi AT %QB56 : WORD;
	.Sfiht1To_Hmi AT %QB58 : WORD;
	.Sfiht2To_Hmi AT %QB60 : WORD;
	.Sfiht3To_Hmi AT %QB62 : WORD;
	.bQRetA_RowStopperMotorFwd AT %QX64.0 : BOOL;	(*  ~ {LinkedWith:TIID^Device 3 (EtherCAT)^Term 1 (EK1100)^Term 9 (EL2809)^Channel 1^Output} *)
	.bQRetA_RowStopperMotorRev AT %QX64.1 : BOOL;	(*  ~ {LinkedWith:TIID^Device 3 (EtherCAT)^Term 1 (EK1100)^Term 9 (EL2809)^Channel 2^Output} *)
	.bQRetB_RowStopperMotorFwd AT %QX64.2 : BOOL;	(*  ~ {LinkedWith:TIID^Device 3 (EtherCAT)^Term 1 (EK1100)^Term 9 (EL2809)^Channel 3^Output} *)
	.bQRetB_RowStopperMotorRev AT %QX64.3 : BOOL;	(*  ~ {LinkedWith:TIID^Device 3 (EtherCAT)^Term 1 (EK1100)^Term 9 (EL2809)^Channel 4^Output} *)
	.bQSpareOutput1 AT %QX64.4 : BOOL;	(*  ~ {LinkedWith:TIID^Device 3 (EtherCAT)^Term 1 (EK1100)^Term 9 (EL2809)^Channel 5^Output} *)
	.bQRetA_WeightOk AT %QX64.5 : BOOL;	(*  ~ {LinkedWith:TIID^Device 3 (EtherCAT)^Term 1 (EK1100)^Term 9 (EL2809)^Channel 6^Output} *)
	.bQRetA_WeightNOk AT %QX64.6 : BOOL;	(*  ~ {LinkedWith:TIID^Device 3 (EtherCAT)^Term 1 (EK1100)^Term 9 (EL2809)^Channel 7^Output} *)
	.bQRetB_WeightOk AT %QX64.7 : BOOL;	(*  ~ {LinkedWith:TIID^Device 3 (EtherCAT)^Term 1 (EK1100)^Term 9 (EL2809)^Channel 8^Output} *)
	.bQRetB_WeightNOk AT %QX65.0 : BOOL;	(*  ~ {LinkedWith:TIID^Device 3 (EtherCAT)^Term 1 (EK1100)^Term 9 (EL2809)^Channel 9^Output} *)
	.bQSpareOutput2 AT %QX65.1 : BOOL;	(*  ~ {LinkedWith:TIID^Device 3 (EtherCAT)^Term 1 (EK1100)^Term 9 (EL2809)^Channel 14^Output} *)
	.bQSpareOutput3 AT %QX65.2 : BOOL;	(*  ~ {LinkedWith:TIID^Device 3 (EtherCAT)^Term 1 (EK1100)^Term 9 (EL2809)^Channel 15^Output} *)
	.bQSpareOutput4 AT %QX65.3 : BOOL;	(*  ~ {LinkedWith:TIID^Device 3 (EtherCAT)^Term 1 (EK1100)^Term 9 (EL2809)^Channel 16^Output} *)
	.bQTowerLampRed AT %QX65.4 : BOOL;	(*  ~ {LinkedWith:TIID^Device 3 (EtherCAT)^Term 1 (EK1100)^Term 9 (EL2809)^Channel 10^Output} *)
	.bQTowerLampGreen AT %QX65.5 : BOOL;	(*  ~ {LinkedWith:TIID^Device 3 (EtherCAT)^Term 1 (EK1100)^Term 9 (EL2809)^Channel 11^Output} *)
	.bQTowerLampYellow AT %QX65.6 : BOOL;	(*  ~ {LinkedWith:TIID^Device 3 (EtherCAT)^Term 1 (EK1100)^Term 9 (EL2809)^Channel 12^Output} *)
	.bQTowerBuzzer AT %QX65.7 : BOOL;	(*  ~ {LinkedWith:TIID^Device 3 (EtherCAT)^Term 1 (EK1100)^Term 9 (EL2809)^Channel 13^Output} *)
	.bQConeFeedingPiston AT %QX66.0 : BOOL;	(*  ~ {LinkedWith:TIID^Device 3 (EtherCAT)^Term 1 (EK1100)^Term 10 (EL2809)^Channel 1^Output} *)
	.bQForwardPiston AT %QX66.1 : BOOL;	(*  ~ {LinkedWith:TIID^Device 3 (EtherCAT)^Term 1 (EK1100)^Term 10 (EL2809)^Channel 2^Output} *)
	.bQReversePiston AT %QX66.2 : BOOL;	(*  ~ {LinkedWith:TIID^Device 3 (EtherCAT)^Term 1 (EK1100)^Term 10 (EL2809)^Channel 3^Output} *)
	.bQTiltingPiston AT %QX66.3 : BOOL;	(*  ~ {LinkedWith:TIID^Device 3 (EtherCAT)^Term 1 (EK1100)^Term 10 (EL2809)^Channel 4^Output} *)
	.bQWrappingPiston1 AT %QX66.4 : BOOL;	(*  ~ {LinkedWith:TIID^Device 3 (EtherCAT)^Term 1 (EK1100)^Term 10 (EL2809)^Channel 5^Output} *)
	.bQWrappingPiston2 AT %QX66.5 : BOOL;	(*  ~ {LinkedWith:TIID^Device 3 (EtherCAT)^Term 1 (EK1100)^Term 10 (EL2809)^Channel 6^Output} *)
	.bQSealingSeparatorYAxisPiston AT %QX66.6 : BOOL;	(*  ~ {LinkedWith:TIID^Device 3 (EtherCAT)^Term 1 (EK1100)^Term 10 (EL2809)^Channel 7^Output} *)
	.bQSealingTopPiston AT %QX66.7 : BOOL;	(*  ~ {LinkedWith:TIID^Device 3 (EtherCAT)^Term 1 (EK1100)^Term 10 (EL2809)^Channel 8^Output} *)
	.bQSealingBottomPiston AT %QX67.0 : BOOL;	(*  ~ {LinkedWith:TIID^Device 3 (EtherCAT)^Term 1 (EK1100)^Term 10 (EL2809)^Channel 9^Output} *)
	.bQSealingSeparatorXAxisPiston AT %QX67.1 : BOOL;	(*  ~ {LinkedWith:TIID^Device 3 (EtherCAT)^Term 1 (EK1100)^Term 10 (EL2809)^Channel 10^Output} *)
	.bQFilmRollerMotor1 AT %QX67.2 : BOOL;	(*  ~ {LinkedWith:TIID^Device 3 (EtherCAT)^Term 1 (EK1100)^Term 10 (EL2809)^Channel 11^Output} *)
	.bQFilmRollerMotor2 AT %QX67.3 : BOOL;	(*  ~ {LinkedWith:TIID^Device 3 (EtherCAT)^Term 1 (EK1100)^Term 10 (EL2809)^Channel 12^Output} *)
	.bQConeCountPiston AT %QX67.4 : BOOL;	(*  ~ {LinkedWith:TIID^Device 3 (EtherCAT)^Term 1 (EK1100)^Term 10 (EL2809)^Channel 13^Output} *)
	.bQFeedingConveyorMotor AT %QX67.5 : BOOL;	(*  ~ {LinkedWith:TIID^Device 3 (EtherCAT)^Term 1 (EK1100)^Term 10 (EL2809)^Channel 14^Output} *)
	.bQWappingConveyorMotor AT %QX67.6 : BOOL;	(*  ~ {LinkedWith:TIID^Device 3 (EtherCAT)^Term 1 (EK1100)^Term 10 (EL2809)^Channel 15^Output} *)
	.bQSealingConveyorMotor AT %QX67.7 : BOOL;	(*  ~ {LinkedWith:TIID^Device 3 (EtherCAT)^Term 1 (EK1100)^Term 10 (EL2809)^Channel 16^Output} *)
	.bQSpareOutput5 AT %QX68.0 : BOOL;	(*  ~ {LinkedWith:TIID^Device 3 (EtherCAT)^Term 1 (EK1100)^Term 12 (EL2008)^Channel 1^Output} *)
	.bQSpareOutput6 AT %QX68.1 : BOOL;	(*  ~ {LinkedWith:TIID^Device 3 (EtherCAT)^Term 1 (EK1100)^Term 12 (EL2008)^Channel 2^Output} *)
	.bQSpareOutput7 AT %QX68.2 : BOOL;	(*  ~ {LinkedWith:TIID^Device 3 (EtherCAT)^Term 1 (EK1100)^Term 12 (EL2008)^Channel 3^Output} *)
	.bQSpareOutput8 AT %QX68.3 : BOOL;	(*  ~ {LinkedWith:TIID^Device 3 (EtherCAT)^Term 1 (EK1100)^Term 12 (EL2008)^Channel 4^Output} *)
	.bQSpareOutput9 AT %QX68.4 : BOOL;	(*  ~ {LinkedWith:TIID^Device 3 (EtherCAT)^Term 1 (EK1100)^Term 12 (EL2008)^Channel 5^Output} *)
	.bQSpareOutput10 AT %QX68.5 : BOOL;	(*  ~ {LinkedWith:TIID^Device 3 (EtherCAT)^Term 1 (EK1100)^Term 12 (EL2008)^Channel 6^Output} *)
	.bQSpareOutput11 AT %QX68.6 : BOOL;	(*  ~ {LinkedWith:TIID^Device 3 (EtherCAT)^Term 1 (EK1100)^Term 12 (EL2008)^Channel 7^Output} *)
	.bQSpareOutput12 AT %QX68.7 : BOOL;	(*  ~ {LinkedWith:TIID^Device 3 (EtherCAT)^Term 1 (EK1100)^Term 12 (EL2008)^Channel 8^Output} *)
	.bQColumnStopperPiston AT %QX69.0 : BOOL;	(*  ~ {LinkedWith:TIID^Device 3 (EtherCAT)^Term 1 (EK1100)^Term 11 (EL2809)^Channel 1^Output} *)
	.bQColumnReversePiston AT %QX69.1 : BOOL;	(*  ~ {LinkedWith:TIID^Device 3 (EtherCAT)^Term 1 (EK1100)^Term 11 (EL2809)^Channel 2^Output} *)
	.bQSeparatorplatePiston AT %QX69.2 : BOOL;	(*  ~ {LinkedWith:TIID^Device 3 (EtherCAT)^Term 1 (EK1100)^Term 11 (EL2809)^Channel 3^Output} *)
	.bQConePusher1Piston AT %QX69.3 : BOOL;	(*  ~ {LinkedWith:TIID^Device 3 (EtherCAT)^Term 1 (EK1100)^Term 11 (EL2809)^Channel 4^Output} *)
	.bQConePusher2Piston AT %QX69.4 : BOOL;	(*  ~ {LinkedWith:TIID^Device 3 (EtherCAT)^Term 1 (EK1100)^Term 11 (EL2809)^Channel 5^Output} *)
	.bQBagPusherForwardPiston AT %QX69.5 : BOOL;	(*  ~ {LinkedWith:TIID^Device 3 (EtherCAT)^Term 1 (EK1100)^Term 11 (EL2809)^Channel 6^Output} *)
	.bQBagPusherReversePiston AT %QX69.6 : BOOL;	(*  ~ {LinkedWith:TIID^Device 3 (EtherCAT)^Term 1 (EK1100)^Term 11 (EL2809)^Channel 7^Output} *)
	.bQBagHolderpiston AT %QX69.7 : BOOL;	(*  ~ {LinkedWith:TIID^Device 3 (EtherCAT)^Term 1 (EK1100)^Term 11 (EL2809)^Channel 8^Output} *)
	.bQBagUp_Down180piston AT %QX70.0 : BOOL;	(*  ~ {LinkedWith:TIID^Device 3 (EtherCAT)^Term 1 (EK1100)^Term 11 (EL2809)^Channel 9^Output} *)
	.bQBagUp_Down50piston AT %QX70.1 : BOOL;	(*  ~ {LinkedWith:TIID^Device 3 (EtherCAT)^Term 1 (EK1100)^Term 11 (EL2809)^Channel 10^Output} *)
	.bQBagTiltingpistonForward AT %QX70.2 : BOOL;	(*  ~ {LinkedWith:TIID^Device 3 (EtherCAT)^Term 1 (EK1100)^Term 11 (EL2809)^Channel 11^Output} *)
	.bQBagTiltingpistonReverse AT %QX70.3 : BOOL;	(*  ~ {LinkedWith:TIID^Device 3 (EtherCAT)^Term 1 (EK1100)^Term 11 (EL2809)^Channel 12^Output} *)
	.bQBagRowHolderpiston AT %QX70.4 : BOOL;	(*  ~ {LinkedWith:TIID^Device 3 (EtherCAT)^Term 1 (EK1100)^Term 11 (EL2809)^Channel 13^Output} *)
	.bQSpareOutput13 AT %QX70.5 : BOOL;	(*  ~ {LinkedWith:TIID^Device 3 (EtherCAT)^Term 1 (EK1100)^Term 11 (EL2809)^Channel 14^Output} *)
	.bQSpareOutput14 AT %QX70.6 : BOOL;	(*  ~ {LinkedWith:TIID^Device 3 (EtherCAT)^Term 1 (EK1100)^Term 11 (EL2809)^Channel 15^Output} *)
	.bQSpareOutput15 AT %QX70.7 : BOOL;	(*  ~ {LinkedWith:TIID^Device 3 (EtherCAT)^Term 1 (EK1100)^Term 11 (EL2809)^Channel 16^Output} *)
END_VAR

(* Data type *)
TYPE ProductionData_PrintData :
STRUCT
	Print:STRING;
	ConeType1:STRING;
	Blend1:STRING;
	DefaultnetWt1:STRING;
	DefaultGrossWt1:STRING;
	LotNo1:STRING;
	BagNo1:STRING;
	Shade1:STRING;
END_STRUCT
END_TYPE

(* Data type *)
TYPE ProductionData_ReportData :
STRUCT
	SERIALNO			:STRING;
	SDATE				:STRING;
	STIME				:STRING;
	BAGNO				:STRING;
	COUNTCODE		:STRING;
	LOTNO				:STRING;
	DFLTNETWEIGHT	:STRING;
	ACTNETWEIGHT		:STRING;
	DFLTGROSSWEIGHT	:STRING;
	ACTGROSSWEIGHT	:STRING;
END_STRUCT
END_TYPE

(* POU MAIN, ST *)
PROGRAM MAIN
	VAR

END_VAR
					(*START / STOP / PAUSE / RESUME*)


	IF (bIMcStartPb OR Start_TapHmi)  AND bAutoModeOn  THEN
	 bMcStartInAuto:=TRUE;
	bMcStopEnable:=FALSE;
	END_IF

	IF  bIMcStopPb OR Stop_TapHmi  OR NOT bAutoModeOn OR NOT bIEmergencySwitchPb THEN
	 bMcStartInAuto:=FALSE;bMcStopEnable:=TRUE;bMcStopEnable1:=TRUE;
	ELSE bMcStopEnable1:=FALSE;
	 END_IF

	IF Pause_TapHmi THEN
	bPauseSeq:=TRUE;END_IF
	IF Resume_TapHmi THEN
	bPauseSeq:=FALSE;END_IF

	IF bIResetPb OR Reset_TapHmi  OR bIResetSealingPb THEN
	bErrorReset:=TRUE;
	ELSE bErrorReset:=FALSE;END_IF

					(*============== Auto/Manual Mode Selection Logic========================*)

		IF bIAutoManualSwitch THEN
			bAutoModeOn:=TRUE; bManualModeOn:=FALSE;
		ELSIF  NOT bIAutoManualSwitch  THEN
			bManualModeOn:=TRUE; bAutoModeOn:=FALSE;
		END_IF

		IF bManualModeOn THEN sMcStatus:='Machine in Manual Mode';
		ELSIF bAutoModeOn THEN sMcStatus:='Machine in Auto Mode';
		END_IF

	IF bMcStartInAuto  AND NOT  bIAutoManualSwitch THEN
	bHidePopUp:=TRUE; END_IF

	IF NOT  bMcStartInAuto  AND NOT  bIAutoManualSwitch THEN
	bManualmode:=TRUE;  END_IF

	IF bHidePopUp AND bManualModeOk_TapHmi THEN
	bManualmode:=TRUE;bAutoModeOn:=FALSE;bHidePopUp:=FALSE; END_IF

	IF bHidePopUp AND bManualModeNOk_TapHmi THEN
	bHidePopUp:=FALSE; END_IF

					 (*====================Logic for Model Selection===============*)

		IF bAutoModeOn AND BagSelect_TapHmi AND NOT bAMainIntStarted THEN
		bABoxModeSelected:=FALSE;BoxSelect_TapHmi:=FALSE;bABagModeSelected:=TRUE; BoxSelect_TapHmi:=FALSE;
		ELSIF bAutoModeOn AND   BoxSelect_TapHmi AND NOT bAMainIntStarted THEN
		bABagModeSelected:=FALSE; BagSelect_TapHmi:=FALSE;bABoxModeSelected:=TRUE;
		END_IF

		IF bABagModeSelected THEN sPackingModeStatus:=' Bag Packing Selected '; END_IF
		IF bABoxModeSelected THEN sPackingModeStatus:=' Carton Packing Selected  '; END_IF




			(****************DATE AND TIME***********)

(*======================= RTC==============================*)

FB_DateTime_1(NET_ID:='5.69.70.240.1.1 ' , DATE_TIME=> );

IF FB_DateTime_1.FBLTIME.systemTime.wHour >0 AND  FB_DateTime_1.FBLTIME.systemTime.wHour<9 THEN
sHourPreFix:='0';sHou:=CONCAT(STR1:=sHourPreFix, Str2:=WORD_TO_STRING(FB_DateTime_1.FBLTIME.systemTime.wHour));
ELSIF FB_DateTime_1.FBLTIME.systemTime.wHour >=10 AND  FB_DateTime_1.FBLTIME.systemTime.wHour<=24 THEN
sHou:=WORD_TO_STRING(FB_DateTime_1.FBLTIME.systemTime.wHour);
END_IF

IF FB_DateTime_1.FBLTIME.systemTime.wDay >0 AND  FB_DateTime_1.FBLTIME.systemTime.wDay<10 THEN
sDayPreFix:='0';sDay:=CONCAT(STR1:=sDayPreFix, Str2:=WORD_TO_STRING(FB_DateTime_1.FBLTIME.systemTime.wDay));
ELSIF FB_DateTime_1.FBLTIME.systemTime.wDay >=10 AND  FB_DateTime_1.FBLTIME.systemTime.wDay<=31 THEN
sDay:=WORD_TO_STRING(FB_DateTime_1.FBLTIME.systemTime.wDay);
END_IF

IF FB_DateTime_1.FBLTIME.systemTime.wMonth >0 AND  FB_DateTime_1.FBLTIME.systemTime.wMonth<10 THEN
sMonthPreFix:='0';sMonth:=CONCAT(STR1:=sMonthPreFix, Str2:=WORD_TO_STRING(FB_DateTime_1.FBLTIME.systemTime.wMonth));
ELSIF FB_DateTime_1.FBLTIME.systemTime.wMonth >=10 AND  FB_DateTime_1.FBLTIME.systemTime.wMonth<=12 THEN
sMonth:=WORD_TO_STRING(FB_DateTime_1.FBLTIME.systemTime.wMonth);
END_IF

sDayF1:=CONCAT(STR1:=sDay, STR2:=':');
sMonthF1:=CONCAT(STR1:=sMonth, STR2:=':');
sDayMonth1:=CONCAT(STR1:=sDayF1, STR2:=sMonthF1);
sDayMonthYear1:=CONCAT(STR1:=sDayMonth1, STR2:=WORD_TO_STRING(FB_DateTime_1.FBLTIME.systemTime.wYear));

sDaateReport:=(sDayMonthYear1);

sDayF:=CONCAT(STR1:=sDay, STR2:='_');
sMonthF:=CONCAT(STR1:=sMonth, STR2:='_');
sDayMonth:=CONCAT(STR1:=sDayF, STR2:=sMonthF);
sDayMonthYear:=CONCAT(STR1:=sDayMonth, STR2:=WORD_TO_STRING(FB_DateTime_1.FBLTIME.systemTime.wYear));

ReportPath:=CONCAT(STR1:='ProductionData', STR2:='_');
ReportPath_Final:=CONCAT(STR1:=ReportPath, STR2:=sDayMonthYear);

ReportPath_Final_1:=CONCAT(STR1:='\\computer-PC\Reports\', STR2:=ReportPath_Final);
ReportPath_Final_2:=CONCAT(STR1:=ReportPath_Final_1, STR2:='.csv');

sDayF1:=CONCAT(STR1:=sDay, STR2:=':');
sMonthF1:=CONCAT(STR1:=sMonth, STR2:=':');
sDayMonth1:=CONCAT(STR1:=sDayF1, STR2:=sMonthF1);
sDayMonthYear1:=CONCAT(STR1:=sDayMonth1, STR2:=WORD_TO_STRING(FB_DateTime_1.FBLTIME.systemTime.wYear));

sDateReport:=(sDayMonthYear1);

sDayF:=CONCAT(STR1:=sDay, STR2:='_');
sMonthF:=CONCAT(STR1:=sMonth, STR2:='_');
sDayMonth:=CONCAT(STR1:=sDayF, STR2:=sMonthF);
sDayMonthYear:=CONCAT(STR1:=sDayMonth, STR2:=WORD_TO_STRING(FB_DateTime_1.FBLTIME.systemTime.wYear));

ReportPathError:=CONCAT(STR1:='ErrorData', STR2:='_');
ReportPath_FinalError:=CONCAT(STR1:=ReportPathError, STR2:=sDayMonthYear);

ReportPath_Final_1Error:=CONCAT(STR1:='\\computer-PC\Reports\', STR2:=ReportPath_FinalError);
ReportPath_Final_2Error:=CONCAT(STR1:=ReportPath_Final_1Error, STR2:='.csv');

DateTimeVar:=FB_DateTime_1.DATE_TIME;



					(*===============Shift Calculation============*)


IF FB_DateTime_1.FBLTIME.systemTime.wHour >= Sfiht1From_Hmi AND FB_DateTime_1.FBLTIME.systemTime.wHour<=Sfiht1To_Hmi THEN
bAShift1Hour:=TRUE;
ELSE
bAShift1Hour:=FALSE;
END_IF



IF FB_DateTime_1.FBLTIME.systemTime.wHour>=Sfiht2From_Hmi AND FB_DateTime_1.FBLTIME.systemTime.wHour <= Sfiht2To_Hmi THEN

bAShift2Hour:=TRUE;
ELSE
bAShift2Hour:=FALSE;
END_IF


IF FB_DateTime_1.FBLTIME.systemTime.wHour>=  Sfiht3From_Hmi AND FB_DateTime_1.FBLTIME.systemTime.wHour<=  Sfiht3To_Hmi THEN

bAShift3Hour:=TRUE;
ELSE
bAShift3Hour:=FALSE;
END_IF

IF bAShift1Hour THEN sShitStatus:='SHIFT - 1';
ELSIF bAShift2Hour THEN sShitStatus:='SHIFT - 2';
ELSIF bAShift3Hour THEN sShitStatus:='SHIFT - 3';
END_IF

Bag_Unit();
ConeFeedCon();
ConeFeedPiston();
Forward_Reverse_Piston();
Ret_A();
Ret_B();
Sealing_Unit();
Tilting_Piston();
Wrapping_Unit();
ErrorData_Report();
Print_Report();
ProductionData_Report();
Bag_Int();
ConeFeedCon_Int();
ConeTransfer_Int();
Main_Int();
Ret_Int();
Sealing_Int();
Wrapping_Int();
Manual();
Weight_Read();
Piston_Alarms();
Outputs();
FilmRollerMotor();
END_PROGRAM

(* POU Auto/Bag_Unit, ST *)
PROGRAM Bag_Unit
VAR
	step: INT;
	iBagRowCounter_243: INT;
	TON_ConeFeedFwdOffDly_1_243: TON;
	TON_Count_243: TON;
	TON_ConePusherOffDly_243: TON;
	TON_ConeFeedFwdOffDly_243: TON;
	TON_ConePusherOnDly_243: TON;
	TON_ConePusherOffDly_2_243: TON;
	TON_ConeFeedFwdOffDly_3_243: TON;
	TON_ConePusherOnDly_2_243: TON;
	TON_ConePusherOnDly_3_243: TON;
	TON_bagPusher_243: TON;
	BagTilting_Blink2_243: TON;
	BagTilting_Blink1_243: TON;

END_VAR
CASE step OF

0:IF IntAllOver AND bABagModeSelected THEN iBagRowCounter_243:= 0; step:=step+1;END_IF

1:	iBagRowCounter_243:= 0; step:=step+1;

2:	bQAColumnConeReversePiston:=FALSE;
	IF bIColumnReversePistonHome AND NOT bPauseSeq THEN
	TON_ConeFeedFwdOffDly_1_243(IN:=FALSE); step := step +1;END_IF

3:	TON_ConeFeedFwdOffDly_1_243(IN:=TRUE , PT:=t#0.1s , Q=> , ET=> );
	IF  TON_ConeFeedFwdOffDly_1_243.Q THEN step := step +1;END_IF

4:	TON_ConeFeedFwdOffDly_1_243(IN:=FALSE);bQAColumnStopperPiston:=TRUE;
	IF  bIColumnStopperPistonEnd AND NOT bPauseSeq THEN
		 bABagOperationStarted_243:= FALSE;bABagUnitRdy_243:=TRUE;
		step := step +1;
	END_IF

5:	IF bABagOperationRdy_243  AND NOT bPauseSeq THEN
	 iBagRowCounter_243:=iBagRowCounter_243+1;bABagOperationStarted_243:=TRUE;
	bABagOperationRdy_243:=FALSE; step:=step+1;
	END_IF

6:	TON_Count_243(IN:=FALSE);bABagOperationRdy_243:=FALSE;
	IF (iBagRowCounter_243 = 1 OR iBagRowCounter_243= 2 OR iBagRowCounter_243 = 3 OR iBagRowCounter_243 = 4 ) AND NOT bPauseSeq THEN
	step:=step+1;

	ELSIF  ( iBagRowCounter_243 = 5 OR  iBagRowCounter_243 = 6 OR  iBagRowCounter_243 = 7 OR iBagRowCounter_243 = 8 ) AND NOT bPauseSeq THEN
	step := 19;
	END_IF

7:	IF   bISeperatorPlatePistonHome AND bIConePusher1PistonHome AND bIBagPusherPistonHome AND bIBagUpDown50PistonEnd
	AND bIBagUpDown180PistonEnd AND bIColumnStopperPistonEnd AND NOT bQABagHolder  AND NOT bPauseSeq THEN
	bQAConePusher2Piston:=FALSE;
	step := step +1;
	END_IF

8:	TON_ConePusherOffDly_243(IN:=TRUE , PT:=t#1s , Q=> , ET=> );
	IF TON_ConePusherOffDly_243.Q  AND NOT bPauseSeq  THEN
	bQAColumnReversePiston:=TRUE;
	TON_ConeFeedFwdOffDly_243(IN:=TRUE , PT:=t#0.1s , Q=> , ET=> );
	IF  TON_ConeFeedFwdOffDly_243.Q AND  bIColumnReversePistonEnd THEN step := step +1;END_IF
	END_IF

9:	TON_ConePusherOffDly_243(IN:=FALSE);
	IF  NOT bPauseSeq  THEN bQAColumnStopperPiston:=FALSE;step := step +1;END_IF

10:	TON_ConeFeedFwdOffDly_243(IN:=FALSE);
	IF bIColumnStopperPistonHome AND NOT bPauseSeq  THEN TON_ConePusherOnDly_243(IN:=TRUE , PT:=t#0.2s , Q=> , ET=> );
	IF TON_ConePusherOnDly_243.Q AND NOT bPauseSeq THEN
 		bQAConePusher1Piston:= TRUE ;bQAColumnReversePiston:=FALSE;step := step +1;
	END_IF END_IF

11: TON_ConePusherOnDly_243(IN:=FALSE);
	 IF bIConePusher1PistonEnd AND bIColumnReversePistonHome AND NOT bPauseSeq THEN
		bQAConePusher2Piston:= TRUE;bABagHalfOpCom_243:=TRUE;step := step +1;
	END_IF

12:	TON_ConePusherOnDly_243(IN:=TRUE , PT:=t#1.5s , Q=> , ET=> );
	IF TON_ConePusherOnDly_243.Q  AND NOT bPauseSeq  THEN bQAConePusher1Piston:= FALSE;
			step := step +1;
	END_IF

13:	TON_ConePusherOnDly_243(IN:=FALSE);
	 IF bIConePusher1PistonHome AND  (iBagRowCounter_243 = 1 OR iBagRowCounter_243 = 2  OR  iBagRowCounter_243 = 3 )
	AND NOT bQABagHolder  AND NOT bPauseSeq THEN
	bQAColumnStopperPiston:=TRUE;
		IF bIColumnStopperPistonEnd AND NOT bPauseSeq THEN
		 bABagOperationStarted:= FALSE;bABagOperationComplete:=TRUE;
		step := 2;END_IF

		ELSIF bIConePusher1PistonHome AND iBagRowCounter_243 =4  AND NOT bQABagHolder  AND NOT bPauseSeq THEN bQAColumnStopperPiston:=FALSE;
		IF  bIColumnStopperPistonHome AND NOT bPauseSeq THEN
		bABagOperationStarted_243:= FALSE;bABagOperationComplete_243:=TRUE;
		step :=14 ;END_IF
	END_IF

14:	step := step +1;

15:	IF   bISeperatorPlatePistonHome AND  bIConePusher1PistonHome AND bIBagPusherPistonHome AND NOT bPauseSeq AND NOT bQABagHolder THEN
	bQABagUp_Down180piston:=FALSE; step := step+1;bQAColumnStopperPiston:=TRUE;

	END_IF

16:	 IF bIBagUpDown180PistonHome AND bISeperatorPlatePistonHome AND bIConePusher1PistonHome AND NOT bQABagHolder  AND NOT bPauseSeq THEN
	bQASeparatorplatePiston:= TRUE ;bQABagUp_Down50piston:=FALSE;step := step +1;
	END_IF

17:	 IF bISeperatorPlatePistonEnd AND bIConePusher1PistonHome AND bIBagPusherPistonHome AND bIBagUpDown180PistonHome
	AND bIColumnStopperPistonEnd AND NOT bQABagHolder  AND NOT bPauseSeq THEN
	bQABagTiltingpistonForward:=TRUE;bQABagBagUp_Down50piston:=TRUE;bQABagTiltingpistonReverse:=FALSE;
	step := step +1;END_IF

18:	bQAColumnStopperPiston:=TRUE;
	 IF bISeperatorPlatePistonEnd AND bIConePusher1PistonHome AND bIBagPusherPistonHome AND bIBagUpDown50PistonEnd AND bIColumnStopperPistonEnd
	AND NOT bQABagHolder  AND NOT bPauseSeq THEN
	step := 2;END_IF

19:	bQAConePusher2Piston:= FALSE;step := step +1;


20:	TON_ConePusherOffDly_2_243(IN:=TRUE , PT:=t#1s , Q=> , ET=> );
	IF TON_ConePusherOffDly_2_243.Q  AND NOT bPauseSeq  THEN step := step +1;
	END_IF

21:	TON_ConePusherOffDly_2_243(IN:=FALSE);
	 IF bISeperatorPlatePistonEnd AND bIConePusher1PistonHome AND bIBagPusherPistonHome AND
	bIBagUpDown50PistonEnd AND bIColumnStopperPistonEnd AND
	bIColumnReversePistonHome AND NOT bQABagHolder  AND NOT bPauseSeq THEN
	bQAColumnReversePiston:=TRUE;step := step +1;END_IF

22:	TON_ConeFeedFwdOffDly_3_243(IN:=TRUE , PT:=t#0.1s , Q=> , ET=> );
	IF  TON_ConeFeedFwdOffDly_3_243.Q AND  bIColumnReversePistonEnd THEN step := step +1;END_IF

23:	TON_ConeFeedFwdOffDly_3_243(IN:=FALSE);bQAColumnStopperPiston:=FALSE;step := step +1;

24:	IF bIColumnStopperPistonHome AND NOT bPauseSeq  THEN TON_ConePusherOnDly_2_243(IN:=TRUE , PT:=t#0.2s , Q=> , ET=> );
	IF TON_ConePusherOnDly_2_243.Q AND NOT bPauseSeq THEN
	bQAConePusher1Piston:= TRUE ;bQAColumnReversePiston:=FALSE;step := step +1;
	END_IF END_IF
25:	TON_ConePusherOnDly_2_243(IN:=FALSE);
	 IF bIConePusher1PistonEnd AND bIColumnReversePistonHome AND NOT bQABagHolder  AND NOT bPauseSeq THEN
	bQAConePusher2Piston:= TRUE;bABagHalfOpCom_243:=TRUE;step := step +1;
	END_IF

26:	TON_ConePusherOnDly_3_243(IN:=TRUE , PT:=t#1.5s , Q=> , ET=> );
	IF TON_ConePusherOnDly_3_243.Q  AND NOT bPauseSeq  THEN
			step := step +1;
	END_IF

27:TON_ConePusherOnDly_3_243(IN:=FALSE);
	 IF bIConePusher1PistonEnd AND (iBagRowCounter_243 = 5 OR iBagRowCounter_243 = 6 OR iBagRowCounter_243 = 7  )
	AND NOT bQABagHolder  AND NOT bPauseSeq THEN
	bQAConePusher1Piston:= FALSE;step := step +1;
	ELSIF
	 bIConePusher1PistonEnd AND iBagRowCounter_243 = 8  AND NOT bQABagHolder  AND NOT bPauseSeq THEN
	step := 29;
	END_IF

28:IF  bIConePusher1PistonHome AND bIColumnStopperPistonHome THEN  bQAColumnStopperPiston:=TRUE;
	bABagOperationStarted_243:= FALSE; bABagOperationComplete_243:=TRUE;
	step := 2;END_IF

29: IF bIConePusher1PistonEnd AND bIBagUpDown50PistonEnd   AND NOT  bQABagHolder AND NOT bPauseSeq THEN
	bQABagPusherForwardPiston:=TRUE;bQABagPusherReversePiston:=FALSE;step := step +1;END_IF

30:TON_bagPusher_243(IN:=TRUE , PT:=t#0.4s , Q=> , ET=> );
	IF (TON_bagPusher_243.Q OR bIBagPusherPistonMiddle) THEN bQABagPusherForwardPiston:=FALSE;bQABagPusherReversePiston:=FALSE; step := step +1;END_IF

31:	TON_bagPusher_243(IN:=FALSE);
	bQABagPusherForwardPiston:=FALSE;bQABagPusherReversePiston:=FALSE;step := step +1;(*END_IF*)

32:	IF NOT bQABagHolder AND NOT bPauseSeq THEN bQASeparatorplatePiston:= FALSE;step := step +1;END_IF

33:	 IF   bISeperatorPlatePistonHome AND NOT bQABagHolder AND NOT bPauseSeq THEN
	 bQAConePusher1Piston:= FALSE;BagOpCom_243:=TRUE;step := step +1;END_IF

34:	IF   bIConePusher1PistonHome AND NOT bPauseSeq THEN
	bQAColumnStopperPiston:=TRUE;
	IF  bIColumnStopperPistonEnd THEN bABagOperationStarted_243:= FALSE;
	bABagOperationComplete_243:=TRUE;bQABagPusherReversePiston:=TRUE;step := step +1;END_IF
	END_IF

35:  IF   bISeperatorPlatePistonHome AND bIConePusher1PistonHome AND bIBagPusherPistonHome AND NOT bPauseSeq AND bIBagiltingPistonEnd THEN
	bQABagUp_Down50piston:=FALSE;step := step +1;END_IF

36:	 IF   bISeperatorPlatePistonHome AND bIConePusher1PistonHome AND bIBagPusherPistonHome AND NOT bPauseSeq AND  bIBagiltingPistonEnd AND
	bIBagUpDown180PistonHome AND bIBagUpDown50PistonHome THEN
	bQABagPusherForwardPiston:=TRUE;bQABagPusherReversePiston:=FALSE;
	IF NOT bIBagPusherPistonMiddle OR bErrorReset THEN bForceBagHolder:=TRUE;step := step +1;END_IF
	END_IF

37:	IF bIBagPusherPistonEnd AND  NOT bPauseSeq THEN
	bQABagPusherForwardPiston:=FALSE;bForceBagHolder:=FALSE;
	bQABagPusherReversePiston:=TRUE;step := step +1;END_IF

38:	IF bIBagPusherPistonHome AND  NOT bPauseSeq THEN
	bQABagPusherForwardPiston:=FALSE;bQABagPusherReversePiston:=FALSE;
	bQABagTiltingpistonForward:=FALSE;bABagTiltingRevOk_243:=TRUE;
	bQABagTiltingpistonReverse:=FALSE;
	step := step +1;END_IF

39: 	IF BagTilting_Blink1_243.Q  AND NOT bPauseSeq THEN
	bQABagTiltingpistonForward:=FALSE; bQABagTiltingpistonReverse:=TRUE;
	ELSE bQABagTiltingpistonReverse:=FALSE;
	IF bIBagTiltingPistonHome THEN bQABagTiltingpistonReverse:=FALSE;bABagTiltingRevOk_243:=FALSE;
	BagTilting_Blink1_243(IN:=FALSE);BagTilting_Blink2_243(IN:=FALSE);step:= step +1;END_IF END_IF


40:	IF bIBagTiltingPistonHome AND  NOT bPauseSeq THEN bQABagTiltingpistonForward:=FALSE;bQABagTiltingpistonReverse:=FALSE;
	bQABagUp_Down180piston:=TRUE;bQABagUp_Down50piston:=TRUE;
	step := step +1;END_IF

41:	IF bIBagResetPb THEN bABagComplete:= TRUE;step:=0;END_IF

END_CASE


IF (bIBagHolder_On OR bIBagHolder_On_Hmi ) AND bISeperatorPlatePistonHome AND bIConePusher1PistonHome THEN

bQABagHolder:=TRUE;bQBagHolder:=TRUE;ELSE bQABagHolder:=FALSE;bQBagHolder:=FALSE;END_IF

bQABagHolderpiston:=bQABagHolder;

BagTilting_Blink1_243(IN:=(bABagTiltingRevOk_243 AND NOT bIBagTiltingPistonHome AND NOT BagTilting_Blink1_243.Q)   , PT:=t#0.6s , Q=> , ET=> );
BagTilting_Blink2_243(IN:=BagTilting_Blink1_243.Q , PT:=t#0.9s , Q=> , ET=> );

IF bIBagTiltingPistonHome THEN bQABagTiltingpistonReverse := FALSE;END_IF
END_PROGRAM

(* POU Auto/ConeFeedCon, ST *)
PROGRAM ConeFeedCon
VAR

END_VAR
bQAFeedingConveyorMotor:=bAConeFeedConveyorStart;

IF bAutoModeOn AND NOT bMcStopEnable AND NOT bRConePresentInConeFeedCon AND NOT bAConeFeedConWait AND NOT bPauseSeq THEN
	bAConeFeedConveyorStart:=TRUE;
ELSE bAConeFeedConveyorStart:=FALSE;END_IF




IF 	((IntAllOver AND bIFeedconeStopSensor AND NOT bIConeFeedingPistonHome) OR
	(IntAllOver AND bIFeedconeStopSensor AND bIConeOrientationTopLimitSwitch))  THEN
	bAConeFeedConWait:=TRUE;
	ELSE bAConeFeedConWait:=FALSE;END_IF

IF bMcStopEnable1 OR NOT bAutoModeOn  THEN
bAConeFeedConveyorStart:=FALSE;
bAConeFeedConWait:=FALSE;
bRConePresentInConeFeedCon:=FALSE;
END_IF
END_PROGRAM

(* POU Auto/ConeFeedPiston, ST *)
PROGRAM ConeFeedPiston
VAR
	ConeFeedPis: INT;
	ConeFeedCount: INT;
	R_TRIG_1: R_TRIG;
	TON_1: TON;
	ConeFeedCounter: CTU;

END_VAR
IF IntAllOver  AND bIConeOrientationTopLimitSwitch AND bIConeFeedingPistonHome AND NOT bPauseSeq   THEN
ConeFeedPistonRdy:=TRUE;
ELSE
ConeFeedPistonRdy:=FALSE;
END_IF

CASE ConeFeedCount OF

0:	R_TRIG_1(CLK:=ConeFeedPistonRdy , Q=> );
		IF R_TRIG_1.Q THEN TON_1(IN:= FALSE); ConeFeedCount:=ConeFeedCount+1; END_IF

1:	IF NOT bPauseSeq  THEN   bAConeFeedCount :=TRUE;
		 ConeFeedCount:=ConeFeedCount+1;END_IF

2:	TON_1(IN :=  TRUE  , PT:=t#1s , Q=> , ET=> );
		IF TON_1.Q THEN  ConeFeedCount:=ConeFeedCount+1; END_IF

3:	bAConeFeedCount :=FALSE;ConeFeedCount:=ConeFeedCount+1;

4: 	IF bIConeFeedingPistonEnd THEN
		ConeFeedCount:=ConeFeedCount+1; END_IF

5:	IF bIConeFeedingPistonHome THEN  ConeFeedCount:=0; END_IF

END_CASE


ConeFeedCounter(
	CU:=bAConeFeedCount  ,
	RESET:=bMcStopEnable  ,
	PV:=TotalNoOfCones,
	Q=> ,
	CV=> );


bQAConeFeedPisOn := bAConeFeedPisOn;

CASE ConeFeedPis OF

0:	 IF IntAllOver  AND NOT bPauseSeq AND bAConeTiltingRdy THEN
	ConeFeedCounter.RESET:=FALSE;ConeFeedPis:=ConeFeedPis+1;END_IF

1:	IF bATiltingCylCom AND NOT bPauseSeq  THEN
	ConeFeedPis:=ConeFeedPis+1;END_IF

2:	IF ConeFeedCounter.CV=1 AND bIConeFeedingPistonHome  AND NOT bAConeFeedingPistonHomeRsError
	AND NOT bPauseSeq AND bITiltingHome THEN
	bAConeFeedPisOn:=TRUE;bATiltingCylCom:=FALSE;ConeFeedPis:=ConeFeedPis+1;END_IF

3:	IF  bIConeFeedingPistonEnd  AND  NOT bAConeFeedingPistonEndRsError AND NOT bPauseSeq THEN
		bAConeFeedPisOn:=FALSE;
		Cone1Reached:=TRUE;
		bAConeFeededCount:=bAConeFeededCount+1;
		ConeFeedPis:=ConeFeedPis+1;END_IF

4:	IF ConeFeedCounter.CV=2 AND bIConeFeedingPistonHome AND NOT bAConeFeedingPistonHomeRsError
	AND NOT bPauseSeq AND (bITiltingMiddle OR bITiltingEnd) THEN
	bAConeFeedPisOn:=TRUE;ConeFeedPis:=ConeFeedPis+1;END_IF

5:	IF  bIConeFeedingPistonEnd  AND  NOT bAConeFeedingPistonEndRsError AND NOT bPauseSeq THEN
		bAConeFeedPisOn:=FALSE;
		Cone2Reached:=TRUE;
		bAConeFeededCount:=bAConeFeededCount+1;
		ConeFeedCounter.RESET:=TRUE;
		ConeFeedPis:=ConeFeedPis+1;END_IF

6:	IF bAConeFeededCount = TotalNoOfCones THEN bAConeFeededCount:=bAConeFeededCount+1;
	ELSIF bAConeFeededCount < TotalNoOfCones THEN bAConeFeededCount:=bAConeFeededCount+2;END_IF

7:	bAConeFeededCount:=0;ConeFeedPis:=ConeFeedPis+1;

8:	ConeFeedCounter.RESET:=FALSE;ConeFeedPis:=1;

END_CASE




IF bMcStopEnable1 OR NOT bAutoModeOn  THEN
ConeFeedPistonRdy:=FALSE;
ConeFeedCount:=0;bAConeFeedCount :=FALSE;
ConeFeedPis:=0;bAConeFeededCount:=0;END_IF
END_PROGRAM

(* POU Auto/Forward_Reverse_Piston, ST *)
PROGRAM Forward_Reverse_Piston
VAR
	FwdRevPis: INT;


END_VAR
bQAForwardPistonOn:=bAForwardPistonOn;
bQAReversePistonOn:=bAReversePistonOn;
CASE FwdRevPis OF

0: IF IntAllOver  AND NOT bPauseSeq AND bAWrapRdy THEN
	FwdRevPis:=FwdRevPis+1;END_IF

1:	FwdRevPis:=FwdRevPis+1;

2:	IF bAFwdRevPisRdy AND (bASealConRdy OR bAWrapRdy) AND NOT bPauseSeq THEN
	bAForwardPistonOn:=TRUE;bAReversePistonOn:=TRUE;bASealConRdy:=FALSE;bAWrapRdy:=FALSE;
	bAFwdRevPisRdy:=FALSE;FwdRevPis:=FwdRevPis+1;END_IF

3:	IF bIForwardPistonEnd AND bIReversePistonEnd AND NOT bAForwardPisEndRsError
	AND NOT bAReversePisEndRsError AND NOT bPauseSeq THEN
	bAFwdRevCount:=bAFwdRevCount+2;
	bAForwardPistonOn:=FALSE;bAReversePistonOn:=FALSE;bAWrappingConRdy:=TRUE;
	FwdRevPis:=FwdRevPis+1;END_IF

4:	IF bIForwardPistonHome AND bIReversePistonHome AND NOT bPauseSeq
	AND NOT bAForwardPisHomeRsError AND NOT bAReversePisHomeRsError THEN
	bAFwdRevCom:=TRUE;FwdRevPis:=FwdRevPis+1;END_IF

5:	IF bAFwdRevCount >= TotalNoOfCones THEN bAFwdRevCount:=0;FwdRevPis:=FwdRevPis+1;
	ELSE FwdRevPis:=FwdRevPis+1;END_IF

6: 	FwdRevPis:=1;

END_CASE


IF bMcStopEnable1 OR NOT bAutoModeOn  THEN
FwdRevPis:=0;bAFwdRevCount:=0;bAFwdRevCom:=FALSE;
bAForwardPistonOn:=FALSE;bAReversePistonOn:=FALSE;
bAFwdRevPisRdy:=FALSE;IntAllOver:=FALSE;END_IF
END_PROGRAM

(* POU Auto/Ret_A, ST *)
PROGRAM Ret_A
VAR
	bARetA_RowStopperFwdOn: BOOL;
	bARetA_RowStopperRevOn: BOOL;
	RetA: INT;
	R_TRIG_RetUnitA_Start: R_TRIG;
	bRetUnitA_Start: BOOL;
	TimerOn: BOOL;
	TON_Speed_RetA: TON;
	RetA_BagOpCom_Speed: TIME;
	bUnitARowStopperStarted: BOOL;
	F_TRIG_1: F_TRIG;
	TON_1: TON;
	step1: INT;
	step2: INT;
	TON_2: TON;
	bAUnitAConeCrossing_Count: BOOL;
	F_TRIG_2: F_TRIG;
	TON_3: TON;
	bAUnitAConeCrossing_FwdCount: BOOL;
	TON_4: TON;
	UnitAConeCrossCount: CTU;
	UnitACompleteCheckCount: CTU;
	bAUnitAWeighOk: BOOL;
	bARetA_RowStopperStarted: BOOL;
	bARetB_RowStopperStarted: BOOL;
	sRetAStatus: STRING;
	RetA_MotorStopDly: TON;
	iATotalNoOfCones: INT;
	UnitACompleteCheckCountCV: CTU;
END_VAR
bQARetA_RowStopperMotorFwd:=bARetA_RowStopperFwdOn;
bQARetA_RowStopperMotorRev:=bARetA_RowStopperRevOn;


R_TRIG_RetUnitA_Start(CLK:=bIUnit_AStartPb, Q=> );
IF R_TRIG_RetUnitA_Start.Q THEN bRetUnitA_Start:=TRUE;TimerOn:=TRUE;END_IF


TON_Speed_RetA(IN:=TimerOn , PT:=t#10m , Q=> , ET=> );
IF bABagComplete THEN RetA_BagOpCom_Speed:=TON_Speed_RetA.ET;END_IF



CASE RetA OF
0:	IF bAutoModeOn AND bAUnitAWeighOk  AND bRetUnitA_Start THEN
	UnitAConeCrossCount.RESET:=TRUE;
	UnitACompleteCheckCount.RESET:=TRUE;
	RetA:=RetA+1;END_IF

1:	IF bAutoModeOn AND NOT bARetA_RowStopperStarted AND UnitACompleteCheckCount.CV=0
	AND UnitAConeCrossCount.CV=0  AND bIUnit_A_RowStopperHome AND NOT bPauseSeq THEN
	UnitACompleteCheckCount.RESET:=FALSE;
	RetA:=RetA+1;END_IF

2:	UnitAConeCrossCount.RESET:=FALSE;
	UnitACompleteCheckCount.RESET:=FALSE;
	RetA:=RetA+1;

3:	IF bAutoModeOn AND NOT bPauseSeq AND NOT bARetB_RowStopperStarted THEN
	RetA:=RetA+1;END_IF

4:	RetA:=RetA+1;

5:	IF  bAutoModeOn  AND NOT bPauseSeq THEN
	bARetA_RowStopperFwdOn:=TRUE;
	bARetA_RowStopperStarted:=TRUE;
	sRetAStatus:='Running';
	RetA_MotorStopDly(in:=FALSE);RetA:=RetA+1;END_IF

6:	IF bIUnit_A_ConeDetectionSensor1 OR  bIUnit_A_ConeDetectionSensor2 OR bIUnit_A_ConeDetectionSensor3 OR bIUnit_A_ConeDetectionSensor4 THEN RetA:=RetA+1;
	ELSIF NOT bIUnit_A_ConeDetectionSensor1 AND  NOT bIUnit_A_ConeDetectionSensor2 AND NOT bIUnit_A_ConeDetectionSensor3 AND NOT bIUnit_A_ConeDetectionSensor4 AND bIUnit_A_RowStopperEnd THEN
	RetA:=10;END_IF

7:	RetA_MotorStopDly(IN:=TRUE , PT:=t#1s , Q=> , ET=> );
	IF RetA_MotorStopDly.Q THEN RetA:=RetA+1;
	END_IF

8:	bARetA_RowStopperFwdOn:=FALSE;
	RetA_MotorStopDly(in:=FALSE);
	RetA:=RetA+1;

9:	IF (UnitAConeCrossCount.CV= 4 ) AND NOT  bIUnit_A_RowStopperEnd   THEN
		RetA_MotorStopDly(In:=FALSE);
		RetA:=4;
		ELSIF bIUnit_A_RowStopperEnd THEN
		RetA:=RetA+1;
		END_IF

10:	bARetA_RowStopperFwdOn:=FALSE;
	RetA_MotorStopDly(in:=FALSE);RetA:=RetA+1;

11:	RetA:=RetA+1;

12:	IF  NOT bPauseSeq THEN
	bARetA_RowStopperRevOn:=TRUE;	RetA:=RetA+1;END_IF

13:	IF bIUnit_A_RowStopperMiddle THEN RetA:=RetA+1;
	ELSIF bIUnit_A_RowStopperHome THEN bARetA_RowStopperRevOn:=FALSE; RetA:=RetA+1;END_IF

14:	IF   (UnitACompleteCheckCount.CV=TotalNoOfCones) AND bIUnit_A_RowStopperHome THEN
	bARetA_RowStopperRevOn:=FALSE;
	UnitAConeCrossCount.RESET:=TRUE;
	UnitACompleteCheckCount.RESET:=TRUE;RetA:=RetA+2;
ELSIF
	(UnitACompleteCheckCount.CV<>TotalNoOfCones) AND bIUnit_A_RowStopperHome THEN
	RetA:=RetA+1;END_IF

15:	IF   (UnitACompleteCheckCount.CV=TotalNoOfCones) AND bIUnit_A_RowStopperHome THEN
	bARetA_RowStopperRevOn:=FALSE;
	UnitAConeCrossCount.RESET:=TRUE;
	UnitACompleteCheckCount.RESET:=TRUE;RetA:=RetA+1;END_IF

16:	bARetA_RowStopperStarted:=FALSE;
	RetA:=RetA+1;

17: RetA:=0;

END_CASE

CASE step1 OF

	0:	IF bUnitARowStopperStarted   AND bAutoModeOn  THEN
		F_TRIG_1(CLK:=bIUnit_B_ConeCrossLimitSwitch , Q=> );
		IF F_TRIG_1.Q THEN TON_1(IN:= FALSE); step1:=step1+1; END_IF END_IF


	1:	TON_1(IN:= FALSE); TON_2(IN:= FALSE); step1:=step1+1;

	2:	 bAUnitAConeCrossing_Count :=TRUE;  step1:=step1+1;

	3: 	TON_1(IN:=  TRUE  , PT:=t#100ms,Q=> , ET=> );
		IF TON_1.Q THEN bAUnitAConeCrossing_Count:=FALSE;   step1:=step1+1; END_IF

	4:	IF   bIUnit_B_ConeCrossLimitSwitch   THEN
		TON_2(IN:=  TRUE  , PT:=t#50ms,Q=> , ET=>);
		IF TON_2.Q THEN TON_1(IN:= FALSE);  step1:=step1+1; END_IF END_IF

	5:	TON_2(IN:= FALSE);
		step1:=0;

END_CASE


CASE step2 OF

	0:	IF bUnitARowStopperStarted    AND bAutoModeOn THEN
		F_TRIG_2(CLK:=bIUnit_A_ConeCrossLimitSwitch , Q=> );
		IF F_TRIG_2.Q THEN TON_1(IN:= FALSE); step2:=step2+1; END_IF END_IF


	1:	TON_3(IN:= FALSE);
		TON_4(IN:= FALSE);
		step2:=step2+1;


	2:	 bAUnitAConeCrossing_FwdCount :=TRUE;
		 step2:=step2+1;

	3: 	TON_3(IN:=  TRUE  , PT:=t#100ms,Q=> , ET=> );
		IF TON_3.Q   THEN  bAUnitAConeCrossing_FwdCount:=FALSE;  step2:=step2+1; END_IF

	4:	IF   bIUnit_A_ConeCrossLimitSwitch   THEN
		TON_4(IN:=  TRUE  , PT:=t#50ms,Q=> , ET=>);
		IF TON_4.Q THEN TON_3(IN:= FALSE);  step2:=step2+1; END_IF END_IF

	5:	TON_4(IN:= FALSE);
		step2:=0;

END_CASE

iATotalNoOfCones:=24;


UnitAConeCrossCount(
	CU:= bAUnitAConeCrossing_FwdCount   ,
	RESET:=bMcStopEnable1 ,
	PV:=3 ,
	Q=> ,
	CV=> );


UnitACompleteCheckCount(
	CU:=  bAUnitAConeCrossing_Count   ,
	RESET:=bMcStopEnable1 ,
	PV:=iATotalNoOfCones ,
	Q=> ,
	CV=> );
END_PROGRAM

(* POU Auto/Ret_B, ST *)
PROGRAM Ret_B
VAR
END_VAR
;
END_PROGRAM

(* POU Auto/Sealing_Unit, ST *)
PROGRAM Sealing_Unit
VAR
	sealingCon: INT;
	CTU_SealingConeCount: CTU;
	TON_SealingConOffDly: TON;
	CTU_SealingRevConeCount: CTU;
	TON_SealConeMissTmr: TON;
	SealUnit: INT;
	TON_SealingPisDly: TON;
	TON_SealingDly_Auto: TON;

	bASealingConeRevCountEnable: BOOL;
END_VAR
CASE sealingCon OF

0:	IF IntAllOver AND  bABagModeSelected  AND NOT bPauseSeq THEN  sealingCon:=sealingCon+1;
	ELSIF IntAllOver AND  bABoxModeSelected  AND NOT bPauseSeq THEN  sealingCon:=sealingCon+1;
	END_IF

1:	IF bABagModeSelected  AND NOT bPauseSeq THEN  bASealingConRdy_Bag:=TRUE; sealingCon:=sealingCon+1;
	ELSIF bABoxModeSelected  AND NOT bPauseSeq THEN bASealingConRdy_Box:=TRUE; sealingCon:=sealingCon+1;
	END_IF

2:	IF bABagModeSelected AND NOT bPauseSeq AND bASealingUnitOperationCom AND
	(bABagUnitRdy_243 OR bABagOperationComplete)  THEN sealingCon:=sealingCon+1;
	ELSIF bABoxModeSelected  AND NOT bPauseSeq AND bASealingUnitOperationCom AND
	(bABoxUnitRdy OR bABoxOperationCom) THEN sealingCon:=sealingCon+1;
	END_IF

3:	IF bABagModeSelected AND NOT bPauseSeq AND NOT bASealConeSet1Completed THEN
	bQASealingConFwd1:=TRUE;bASealConeSet1Started:=TRUE;bABagUnitRdy_243:=FALSE;bABagOperationComplete:=FALSE;sealingCon:=sealingCon+1;
	ELSIF bABagModeSelected AND NOT bPauseSeq AND  bASealConeSet1Completed THEN
	bQASealingConFwd2:=TRUE;bASealConeSet2Started:=TRUE;bASealConeSet1Completed:=FALSE;
	bABagUnitRdy_243:=FALSE;bABagOperationComplete:=FALSE;sealingCon:=sealingCon+1;
	ELSIF bABoxModeSelected  AND NOT bPauseSeq THEN
	bQASealingConRev:=TRUE;bABoxUnitRdy:=FALSE;bABoxOperationCom:=FALSE;sealingCon:=sealingCon+3;
	END_IF

4:	IF CTU_SealingConeCount.CV >=2 AND bABagModeSelected AND bQASealingConFwd1 THEN
	sealingCon:=sealingCon+1;
	ELSIF CTU_SealingConeCount.CV >=1 AND bABagModeSelected AND bQASealingConFwd2 THEN
	bQABagRowHolderpiston:=TRUE;sealingCon:=sealingCon+1;
	END_IF

5:	TON_SealingConOffDly(IN:=TRUE , PT:=t#2s , Q=> , ET=> );
	IF TON_SealingConOffDly.Q AND bQASealingConFwd1  THEN
	bQASealingConFwd1:=FALSE;bASealConeSet1Completed:=TRUE;sealingCon:=sealingCon+1;
	ELSIF TON_SealingConOffDly.Q AND bQASealingConFwd2  THEN
	bQASealingConFwd2:=FALSE;bASealConeSet2Completed:=FALSE;bQABagRowHolderpiston:=FALSE;
	bASealConeSet2Completed:=TRUE;sealingCon:=sealingCon+3;
	END_IF

6: 	sealingCon:=sealingCon+1;

7:	IF CTU_SealingRevConeCount.CV >= 2 AND bABoxModeSelected AND bQASealingConRev THEN
	bQASealingConRev:=FALSE;bASealConeRevSetCompleted:=TRUE;sealingCon:=sealingCon+1;END_IF

8:	sealingCon:=1;

	END_CASE

TON_SealConeMissTmr(IN:=(bQASealingConFwd1 OR bQASealingConFwd2 OR bQASealingConRev) , PT:=t#10s , Q=> , ET=> );
IF TON_SealConeMissTmr.Q AND bQASealingConFwd1 THEN bASealConeMissError1:=TRUE;
ELSIF TON_SealConeMissTmr.Q AND bQASealingConFwd2 THEN bASealConeMissError2:=TRUE;
ELSIF TON_SealConeMissTmr.Q AND bQASealingConRev THEN bASealConeMissError3:=TRUE;
END_IF

IF bASealConeMissError1 OR bASealConeMissError2 OR bASealConeMissError3 THEN
bASealConeMissError:=TRUE;bASealConeMissErrorStatus:='Cone Miss In Sealing Conveyor';END_IF

IF bASealConeMissError1 AND bQASealingConFwd1 THEN 	bQASealingConFwd1:=FALSE;
ELSIF bASealConeMissError2 AND bQASealingConFwd2 THEN 	bQASealingConFwd2:=FALSE;
ELSIF bASealConeMissError3 AND bQASealingConRev THEN 	bQASealingConRev:=FALSE;END_IF


IF bASealConeMissError1 AND NOT bPauseSeq AND bErrorReset THEN
	bASealConeMissError1:=FALSE;bQASealingConFwd1:=TRUE;
ELSIF bASealConeMissError2 AND NOT bPauseSeq AND bErrorReset THEN
	bASealConeMissError2:=FALSE;bQASealingConFwd2:=TRUE;
ELSIF bASealConeMissError3 AND NOT bPauseSeq AND bErrorReset THEN
	bASealConeMissError3:=FALSE;bQASealingConRev:=TRUE;
END_IF






IF (bQASealingConFwd1 OR bQASealingConFwd2) AND bIConeCountsensor THEN
	bASealingConeCountEnable:=TRUE;
ELSE bASealingConeCountEnable:=FALSE;END_IF
CTU_SealingConeCount(
	CU:=bASealingConeCountEnable ,
	RESET:= ,
	PV:= ,
	Q=> ,
	CV=> );

IF bQASealingConRev  AND bISpare4 THEN
	bASealingConeRevCountEnable:=TRUE;
ELSE bASealingConeRevCountEnable:=FALSE;END_IF
CTU_SealingRevConeCount(
	CU:=bASealingConeRevCountEnable ,
	RESET:= ,
	PV:= ,
	Q=> , 
	CV=> );


CASE SealUnit OF

0:	IF IntAllOver  AND NOT bPauseSeq AND bASealingUnitInt THEN
	SealUnit:=SealUnit+1;END_IF

1:	SealUnit:=SealUnit+1;

2:	IF bASealUnitStart AND NOT bPauseSeq AND bAutoModeOn  AND WrappingSafety THEN
	bQASealingSeparatorYAxisPiston:=TRUE;SealUnit:=SealUnit+1;END_IF

3:	IF bISealingSeparatorYAxisPistoEnd AND NOT bPauseSeq THEN
	bQASealingTopPiston:=TRUE;bQASealingBottomPiston:=TRUE;SealUnit:=SealUnit+1;END_IF

4:	TON_SealingPisDly(IN:=TRUE , PT:=t#2s , Q=> , ET=> );
	IF (bISealingTopPistonEnd AND bISealingBottomPistonEnd) OR TON_SealingPisDly.Q THEN
	SealUnit:=SealUnit+1;END_IF

5:	TON_SealingDly_Auto(IN:=TRUE , PT:= t#2s, Q=> , ET=> );
	IF TON_SealingDly_Auto.Q THEN SealUnit:=SealUnit+1;END_IF

6:	bQASealingSeparatorXAxisPiston:=TRUE;TON_SealingPisDly(IN:=FALSE);TON_SealingDly_Auto(IN:=FALSE);
	SealUnit:=SealUnit+1;

7:	IF bISealingSeparatorXAxisPistonEnd AND NOT bPauseSeq THEN
	bQASealingSeparatorYAxisPiston:=FALSE;
	bQASealingTopPiston:=FALSE;bQASealingBottomPiston:=FALSE;
	bQASealingSeparatorXAxisPiston:=FALSE;SealUnit:=SealUnit+1;END_IF

8:	IF SealingSafety AND NOT bPauseSeq THEN
	bASealingUnitOperationCom:=TRUE;SealUnit:=SealUnit+1;END_IF

9:	SealUnit:=0;

END_CASE
END_PROGRAM

(* POU Auto/Tilting_Piston, ST *)
PROGRAM Tilting_Piston
VAR
	TiltPis: INT;

END_VAR
CASE TiltPis OF

0: IF IntAllOver  AND NOT bPauseSeq AND bAConeFwdRevRdy THEN
	TiltPis:=TiltPis+1;END_IF

1:	TiltPis:=TiltPis+1;

2:	IF Cone1Reached  AND NOT bPauseSeq AND bIForwardPistonHome AND bIReversePistonHome THEN
	bAConeTiltingCount:=bAConeTiltingCount+1;bATiltingPistonOn:=TRUE;END_IF

3: 	IF bITiltingEnd AND NOT bPauseSeq AND NOT bAConeTiltingPistonEndRsError THEN
	Cone1Reached:=FALSE;TiltPis:=TiltPis+1;END_IF

4:	IF Cone2Reached AND  NOT bPauseSeq THEN
	bAConeTiltingCount:=bAConeTiltingCount+1;bAFwdRevPisRdy:=TRUE;Cone2Reached:=FALSE;TiltPis:=TiltPis+1;END_IF

5:	IF bAFwdRevCom AND NOT bPauseSeq THEN
	bATiltingPistonOn:=FALSE;TiltPis:=TiltPis+1;END_IF

6:	IF bITiltingHome AND NOT bPauseSeq AND NOT bAConeTiltingPistonHomeRsError THEN
	bATiltingCylCom:=TRUE;TiltPis:=TiltPis+1;END_IF

7: IF bAConeTiltingCount >= TotalNoOfCones THEN bAConeTiltingCount := 0;
	ELSE TiltPis:=TiltPis+1;END_IF

8:	TiltPis:=1;

END_CASE

IF bMcStopEnable1 OR NOT bAutoModeOn  THEN
TiltPis:=0;bAConeTiltingCount := 0;bATiltingCylCom:=FALSE;
bAFwdRevPisRdy:=FALSE;Cone2Reached:=FALSE;Cone1Reached:=FALSE;
bATiltingPistonOn:=FALSE;bAConeFwdRevRdy:=FALSE;END_IF
END_PROGRAM

(* POU Auto/Wrapping_Unit, ST *)
PROGRAM Wrapping_Unit
VAR
	WrappingCon: INT;
	WrapPis: INT;

	bASealConRdy: BOOL;
	TON_bAWrapConeAlaign: TON;

	bASheetFeedError1: BOOL;
	bASheetFeedError2: BOOL;
END_VAR
CASE WrappingCon OF
0: 	IF IntAllOver  AND NOT bPauseSeq AND bAWrappingPisCylComInt THEN
	WrappingCon:=WrappingCon+1;END_IF

1:	IF (bAWrappingPisCylCom OR bAWrappingPisCylComInt ) AND NOT bPauseSeq THEN
	bAWrappingConRdy:=FALSE;bAWrappingPisCylCom:=FALSE;
	bAWrappingPisCylComInt:=FALSE;WrappingCon:=WrappingCon+1;END_IF

2:	IF bAWrappingConRdy AND WrappingSafety AND NOT bIWrappingCone1 AND NOT bIWrappingCone2 AND NOT bPauseSeq THEN
	bAWrapConeAlaignError:=FALSE;bAWrappingConRdy:=FALSE;
	sWrappingConStatus:='Continue Machine Runnig';WrappingCon:=WrappingCon+2;

	ELSIF bAWrappingConRdy AND WrappingSafety AND NOT bPauseSeq AND bIWrappingCone1  THEN
	bAWrapConeAlaignError:=TRUE;sWrappingConStatus:='Please Check Wrap Cone 1';WrappingCon:=WrappingCon+1;

	ELSIF bAWrappingConRdy AND WrappingSafety AND NOT bPauseSeq AND bIWrappingCone2  THEN
	bAWrapConeAlaignError:=TRUE;sWrappingConStatus:='Please Check Wrap Cone 2';WrappingCon:=WrappingCon+1;

	ELSIF bAWrappingConRdy AND WrappingSafety AND NOT bPauseSeq AND (bIWrappingCone1 OR bIWrappingCone2)  THEN
	bAWrapConeAlaignError:=TRUE;
	sWrappingConStatus:='Please Check Wrap Cone 1 & 2';WrappingCon:=WrappingCon+1;
	END_IF

3:	IF bErrorReset AND NOT bIWrappingCone1 AND NOT bIWrappingCone2 AND NOT bPauseSeq THEN
	bAWrapConeAlaignError:=FALSE;sWrappingConStatus:='Continue Machine Runnig';WrappingCon:=WrappingCon+1;END_IF

4:	bAWrappingConOn:=TRUE;WrappingCon:=WrappingCon+1;

5:	IF bIWrappingCone1 AND bIWrappingCone2  THEN
	bAWrappingConOn:=FALSE;WrappingCon:=WrappingCon+1;END_IF

6:	IF NOT bAWrapConeAlaignError1 AND NOT bPauseSeq THEN
	bAWrappingPisRdy:=TRUE;bASealConRdy:=TRUE;WrappingCon:=WrappingCon+1;END_IF

7:	WrappingCon:=1;

END_CASE

TON_bAWrapConeAlaign(IN:=bAWrappingConOn , PT:=t#3s , Q=> , ET=> );
IF TON_bAWrapConeAlaign.Q THEN bAWrapConeAlaignError1:=TRUE;END_IF

IF bErrorReset AND bIWrappingCone1 AND bIWrappingCone2 AND bAWrapConeAlaignError1 THEN
bAWrapConeAlaignError1:=FALSE;END_IF


CASE WrapPis OF
0:	IF bAWrappingPisRdy AND NOT bPauseSeq THEN
	bAWrapPiston1On:=TRUE;bAWrapPiston2On:=TRUE;WrapPis:=WrapPis+1;END_IF

1:	bAWrappingPisRdy:=FALSE;WrapPis:=WrapPis+1;

2:	IF bIWrappingChanelPiston1Middle OR bIWrappingChanelPiston2Middle THEN
	WrapPis:=WrapPis+1;END_IF

3:	IF bASealingConRdy AND NOT bPauseSeq THEN
	WrapPis:=WrapPis+2;
	ELSIF NOT bASealingConRdy THEN
	 bAWrapPiston1On:=FALSE;bAWrapPiston2On:=FALSE;WrapPis:=WrapPis+1;END_IF

4:	IF bASealingConRdy AND NOT bPauseSeq THEN
	bAWrapPiston1On:=TRUE;bAWrapPiston2On:=TRUE;WrapPis:=WrapPis+1;END_IF

5: 	IF bIWrappingChanelPiston1End AND bIWrappingChanelPiston2End AND bAFilmLoaded1 AND bAFilmLoaded1
	AND NOT bASheetFeedError AND NOT bAWrapPis1EndRsError AND NOT bAWrapPis2EndRsError
	AND NOT bPauseSeq THEN
	 bAWrapPiston1On:=FALSE;bAWrapPiston2On:=FALSE;WrapPis:=WrapPis+3;
	ELSIF  bIWrappingChanelPiston1End AND bIWrappingChanelPiston2End AND NOT bAFilmLoaded1 THEN  bASheetFeedError1:=TRUE;  WrapPis:=WrapPis+2;
	ELSIF  bIWrappingChanelPiston1End AND bIWrappingChanelPiston2End AND NOT bAFilmLoaded2 THEN bASheetFeedError2:=TRUE;  WrapPis:=WrapPis+2;
	ELSIF bAWrapPis1EndRsError OR bAWrapPis2EndRsError THEN WrapPis:=WrapPis+1;
	END_IF

6:  	IF bErrorReset AND NOT bPauseSeq AND NOT bAWrapPis1EndRsError AND NOT bAWrapPis2EndRsError THEN
	WrapPis:=5;
	END_IF

7:	IF bASheetFeedError1 OR bASheetFeedError2 AND bErrorReset THEN
	bAFilmLoaded1:=TRUE;bAFilmLoaded2:=TRUE;bASheetFeedError1:=FALSE;bASheetFeedError2:=FALSE;	WrapPis:=5;END_IF


8:	bAFilmLoaded1:=FALSE;;bAFilmLoaded2:=FALSE; WrapPis:=WrapPis+1;

9:	IF WrappingSafety AND NOT bPauseSeq THEN
	bAWrappingPisCylCom:=TRUE; bASealUnitStart:=TRUE;WrapPis:=WrapPis+1;END_IF

10:	WrapPis:=0;

END_CASE
END_PROGRAM

(* POU DataLog/ErrorData_Report, ST *)
PROGRAM ErrorData_Report
VAR
END_VAR
;
END_PROGRAM

(* POU DataLog/Print_Report, ST *)
PROGRAM Print_Report
VAR
	step: INT;


	TON_2: TON;
	TON_1: TON;
END_VAR
IF PrintEnable_TogHmi THEN PrintEnabled:=TRUE;PrintValue:=1;ELSE PrintEnabled:=FALSE;PrintValue:=0;END_IF

		ProductionData_PrintData.Print						:=INT_TO_STRING( PrintValue );
		ProductionData_PrintData.ConeType1				:=(COUNT_DIS);
		ProductionData_PrintData.Blend1					:=(BLEND_DIS);
		ProductionData_PrintData.DefaultnetWt1				:=(Actual_NetWeight_Report);
		ProductionData_PrintData.DefaultGrossWt1			:=(Actual_GrossWeight_Report);
		ProductionData_PrintData.LotNo1					:=(LOTNO_DIS);
		ProductionData_PrintData.BagNo1					:=DINT_TO_STRING(CARTONNO_DIS);
		ProductionData_PrintData.Shade1					:=(SHADE_DIS);

		(*	######## Print Data Values		#####	*)

ProductionDataValues_Print:= CONCAT(ProductionData_PrintData.Print,',');
ProductionDataValues_Print:=	 CONCAT( ProductionDataValues_Print,ProductionData_PrintData.ConeType1);
ProductionDataValues_Print:= CONCAT( ProductionDataValues_Print,',');
ProductionDataValues_Print:=	 CONCAT( ProductionDataValues_Print,ProductionData_PrintData.Blend1);
ProductionDataValues_Print:= CONCAT( ProductionDataValues_Print,',');
ProductionDataValues_Print:=	 CONCAT( ProductionDataValues_Print,ProductionData_PrintData.DefaultnetWt1);
ProductionDataValues_Print:= CONCAT( ProductionDataValues_Print,',');
ProductionDataValues_Print:=	 CONCAT( ProductionDataValues_Print,ProductionData_PrintData.DefaultGrossWt1);
ProductionDataValues_Print:= CONCAT( ProductionDataValues_Print,',');
ProductionDataValues_Print:=	 CONCAT( ProductionDataValues_Print,ProductionData_PrintData.LotNo1);
ProductionDataValues_Print:= CONCAT( ProductionDataValues_Print,',');
ProductionDataValues_Print:=	 CONCAT( ProductionDataValues_Print,ProductionData_PrintData.BagNo1);
ProductionDataValues_Print:= CONCAT( ProductionDataValues_Print,',');
ProductionDataValues_Print:=	 CONCAT( ProductionDataValues_Print,ProductionData_PrintData.Shade1);
ProductionDataValues_Print:= CONCAT( ProductionDataValues_Print,'$0A');


					(*	######## Print Data head#####	*)
ProductionData_Print:= CONCAT( 'Print',',');
		ProductionData_Print:=	 CONCAT( ProductionData_Print,'Count Type');
		ProductionData_Print:= CONCAT( ProductionData_Print,',');
ProductionData_Print:=	 CONCAT( ProductionData_Print,'Blend');
		ProductionData_Print:= CONCAT( ProductionData_Print,',');
ProductionData_Print:=	 CONCAT( ProductionData_Print,'NetWt');
		ProductionData_Print:= CONCAT( ProductionData_Print,',');
ProductionData_Print:=	 CONCAT( ProductionData_Print,'Grss Wt');
		ProductionData_Print:= CONCAT( ProductionData_Print,',');
ProductionData_Print:=	 CONCAT( ProductionData_Print,'Lot No');
		ProductionData_Print:= CONCAT( ProductionData_Print,',');
ProductionData_Print:=	 CONCAT( ProductionData_Print,'Bag No');
		ProductionData_Print:= CONCAT( ProductionData_Print,',');
ProductionData_Print:=	 CONCAT( ProductionData_Print,'Shade');
		ProductionData_Print:= CONCAT( ProductionData_Print,'$0A');

FB_FileOpen1(
	sNetId:='192.168.225.76.1.1',
	sPathName:= '\\ACPBAG\Reports\productiondata.csv' ,
	nMode:=FOPEN_MODEAPPEND ,
	ePath:=PATH_GENERIC ,
	bExecute:= ,
	tTimeout:=T#2s ,
	bBusy=> ,
	bError=> ,
	nErrId=> ,
	hFile=> );

FB_FileWrite1(
	sNetId:='192.168.225.76.1.1',
	hFile:=FB_FileOpen1.hFile ,
	pWriteBuff:=ADR(ProductionDataValues_Print_Com),
	cbWriteLen:=LEN(ProductionDataValues_Print_Com),
	bExecute:= ,
	tTimeout:=T#2s ,
	bBusy=> ,
	bError=> ,
	nErrId=> ,
	cbWrite=> );


FB_FileClose1(
	sNetId:='192.168.225.76.1.1',
	hFile:=FB_FileOpen1.hFile ,
	bExecute:= ,
	tTimeout:=T#2s ,
	bBusy=> ,
	bError=> ,
	nErrId=> );

FB_FileDelete1(
	sNetId:='192.168.225.76.1.1',
	sPathName:= '\\ACPBAG\Reports\productiondata.csv' ,
	ePath:=PATH_GENERIC ,
	bExecute:= ,
	tTimeout:=T#2s ,
	bBusy=> ,
	bError=> ,
	nErrId=> );

CASE step OF

0: IF PrintOk THEN
	TON_2(IN:=FALSE);
	FB_FileOpen1.bExecute:=TRUE;
	IF NOT FB_FileOpen1.bBusy AND NOT FB_FileOpen1.bError AND FB_FileOpen1.hFile>0 THEN  step:=step+1;END_IF
	END_IF

1:	IF NOT FB_FileOpen1.bBusy AND NOT FB_FileOpen1.bError AND FB_FileOpen1.hFile>0 THEN  PrintOk:=FALSE;step:=step+1;END_IF

2:
	ProductionDataValues_Print_Com:=ProductionData_Print;
	FB_FileWrite1.bExecute:=TRUE;
	IF NOT FB_FileWrite1.bBusy AND NOT FB_FileWrite1.bError THEN step:=step+1;END_IF

3:	IF NOT FB_FileWrite1.bBusy AND NOT FB_FileWrite1.bError THEN FB_FileWrite1.bExecute:=FALSE; step:=step+1;END_IF

4:	ProductionDataValues_Print_Com:=ProductionDataValues_Print;
	FB_FileWrite1.bExecute:=TRUE;
	IF NOT FB_FileWrite1.bBusy AND NOT FB_FileWrite1.bError THEN step:=step+1;END_IF

5:	step:=step+1;

6:	IF NOT FB_FileWrite1.bBusy AND NOT FB_FileWrite1.bError THEN FB_FileWrite1.bExecute:=FALSE; step:=step+1;END_IF


7:	FB_FileClose1.bExecute:=TRUE;
	 IF NOT FB_FileClose1.bBusy AND NOT FB_FileClose1.bError THEN  step:=step+1;END_IF

8:	TON_1(IN:=TRUE , PT:=t#0.1s , Q=> , ET=> );
	IF TON_1.Q THEN step:=step+1;END_IF

9:	IF NOT FB_FileDelete1.bBusy AND NOT FB_FileDelete1.bError THEN
	TON_1(IN:=FALSE);
	(*FB_FileDelete1.bExecute:=TRUE;*)step:=step+1;END_IF

10:
	FB_FileOpen1.bExecute:=FALSE;
	FB_FileWrite1.bExecute:=FALSE;
	FB_FileClose1.bExecute:=FALSE;
	FB_FileDelete1.bExecute:=FALSE;
	step:=step+1;

11:		TON_2(IN:=TRUE , PT:=t#10s , Q=> , ET=> );
	IF TON_2.Q THEN(* PrintOk:=TRUE;	*) step:=0;END_IF

END_CASE
END_PROGRAM

(* POU Print, ST *)
PROGRAM Print
VAR

	step: INT;


	TON_2: TON;
	TON_1: TON;
END_VAR
IF PrintEnable_TogHmi THEN PrintEnabled:=TRUE;PrintValue:=1;ELSE PrintEnabled:=FALSE;PrintValue:=0;END_IF

		ProductionData_PrintData.Print						:=INT_TO_STRING( PrintValue );
		ProductionData_PrintData.ConeType1				:=(COUNT_DIS);
		ProductionData_PrintData.Blend1					:=(BLEND_DIS);
		ProductionData_PrintData.DefaultnetWt1				:=(Actual_NetWeight_Report);
		ProductionData_PrintData.DefaultGrossWt1			:=(Actual_GrossWeight_Report);
		ProductionData_PrintData.LotNo1					:=(LOTNO_DIS);
		ProductionData_PrintData.BagNo1					:=DINT_TO_STRING(CARTONNO_DIS);
		ProductionData_PrintData.Shade1					:=(SHADE_DIS);

		(*	######## Print Data Values		#####	*)

ProductionDataValues_Print:= CONCAT(ProductionData_PrintData.Print,',');
ProductionDataValues_Print:=	 CONCAT( ProductionDataValues_Print,ProductionData_PrintData.ConeType1);
ProductionDataValues_Print:= CONCAT( ProductionDataValues_Print,',');
ProductionDataValues_Print:=	 CONCAT( ProductionDataValues_Print,ProductionData_PrintData.Blend1);
ProductionDataValues_Print:= CONCAT( ProductionDataValues_Print,',');
ProductionDataValues_Print:=	 CONCAT( ProductionDataValues_Print,ProductionData_PrintData.DefaultnetWt1);
ProductionDataValues_Print:= CONCAT( ProductionDataValues_Print,',');
ProductionDataValues_Print:=	 CONCAT( ProductionDataValues_Print,ProductionData_PrintData.DefaultGrossWt1);
ProductionDataValues_Print:= CONCAT( ProductionDataValues_Print,',');
ProductionDataValues_Print:=	 CONCAT( ProductionDataValues_Print,ProductionData_PrintData.LotNo1);
ProductionDataValues_Print:= CONCAT( ProductionDataValues_Print,',');
ProductionDataValues_Print:=	 CONCAT( ProductionDataValues_Print,ProductionData_PrintData.BagNo1);
ProductionDataValues_Print:= CONCAT( ProductionDataValues_Print,',');
ProductionDataValues_Print:=	 CONCAT( ProductionDataValues_Print,ProductionData_PrintData.Shade1);
ProductionDataValues_Print:= CONCAT( ProductionDataValues_Print,'$0A');


					(*	######## Print Data head#####	*)
ProductionData_Print:= CONCAT( 'Print',',');
		ProductionData_Print:=	 CONCAT( ProductionData_Print,'Count Type');
		ProductionData_Print:= CONCAT( ProductionData_Print,',');
ProductionData_Print:=	 CONCAT( ProductionData_Print,'Blend');
		ProductionData_Print:= CONCAT( ProductionData_Print,',');
ProductionData_Print:=	 CONCAT( ProductionData_Print,'NetWt');
		ProductionData_Print:= CONCAT( ProductionData_Print,',');
ProductionData_Print:=	 CONCAT( ProductionData_Print,'Grss Wt');
		ProductionData_Print:= CONCAT( ProductionData_Print,',');
ProductionData_Print:=	 CONCAT( ProductionData_Print,'Lot No');
		ProductionData_Print:= CONCAT( ProductionData_Print,',');
ProductionData_Print:=	 CONCAT( ProductionData_Print,'Bag No');
		ProductionData_Print:= CONCAT( ProductionData_Print,',');
ProductionData_Print:=	 CONCAT( ProductionData_Print,'Shade');
		ProductionData_Print:= CONCAT( ProductionData_Print,'$0A');

FB_FileOpen1(
	sNetId:='192.168.225.76.1.1',
	sPathName:= '\\ACPBAG\Reports\productiondata.csv' ,
	nMode:=FOPEN_MODEAPPEND ,
	ePath:=PATH_GENERIC ,
	bExecute:= ,
	tTimeout:=T#2s ,
	bBusy=> ,
	bError=> ,
	nErrId=> ,
	hFile=> );

FB_FileWrite1(
	sNetId:='192.168.225.76.1.1',
	hFile:=FB_FileOpen1.hFile ,
	pWriteBuff:=ADR(ProductionDataValues_Print_Com),
	cbWriteLen:=LEN(ProductionDataValues_Print_Com),
	bExecute:= ,
	tTimeout:=T#2s ,
	bBusy=> ,
	bError=> ,
	nErrId=> ,
	cbWrite=> );


FB_FileClose1(
	sNetId:='192.168.225.76.1.1',
	hFile:=FB_FileOpen1.hFile ,
	bExecute:= ,
	tTimeout:=T#2s ,
	bBusy=> ,
	bError=> ,
	nErrId=> );

FB_FileDelete1(
	sNetId:='192.168.225.76.1.1',
	sPathName:= '\\ACPBAG\Reports\productiondata.csv' ,
	ePath:=PATH_GENERIC ,
	bExecute:= ,
	tTimeout:=T#2s ,
	bBusy=> ,
	bError=> ,
	nErrId=> );

CASE step OF

0: IF PrintOk THEN
	TON_2(IN:=FALSE);
	FB_FileOpen1.bExecute:=TRUE;
	IF NOT FB_FileOpen1.bBusy AND NOT FB_FileOpen1.bError AND FB_FileOpen1.hFile>0 THEN  step:=step+1;END_IF
	END_IF

1:	IF NOT FB_FileOpen1.bBusy AND NOT FB_FileOpen1.bError AND FB_FileOpen1.hFile>0 THEN  PrintOk:=FALSE;step:=step+1;END_IF

2:
	ProductionDataValues_Print_Com:=ProductionData_Print;
	FB_FileWrite1.bExecute:=TRUE;
	IF NOT FB_FileWrite1.bBusy AND NOT FB_FileWrite1.bError THEN step:=step+1;END_IF

3:	IF NOT FB_FileWrite1.bBusy AND NOT FB_FileWrite1.bError THEN FB_FileWrite1.bExecute:=FALSE; step:=step+1;END_IF

4:	ProductionDataValues_Print_Com:=ProductionDataValues_Print;
	FB_FileWrite1.bExecute:=TRUE;
	IF NOT FB_FileWrite1.bBusy AND NOT FB_FileWrite1.bError THEN step:=step+1;END_IF

5:	step:=step+1;

6:	IF NOT FB_FileWrite1.bBusy AND NOT FB_FileWrite1.bError THEN FB_FileWrite1.bExecute:=FALSE; step:=step+1;END_IF


7:	FB_FileClose1.bExecute:=TRUE;
	 IF NOT FB_FileClose1.bBusy AND NOT FB_FileClose1.bError THEN  step:=step+1;END_IF

8:	TON_1(IN:=TRUE , PT:=t#0.1s , Q=> , ET=> );
	IF TON_1.Q THEN step:=step+1;END_IF

9:	IF NOT FB_FileDelete1.bBusy AND NOT FB_FileDelete1.bError THEN
	TON_1(IN:=FALSE);
	(*FB_FileDelete1.bExecute:=TRUE;*)step:=step+1;END_IF

10:
	FB_FileOpen1.bExecute:=FALSE;
	FB_FileWrite1.bExecute:=FALSE;
	FB_FileClose1.bExecute:=FALSE;
	FB_FileDelete1.bExecute:=FALSE;
	step:=step+1;

11:		TON_2(IN:=TRUE , PT:=t#10s , Q=> , ET=> );
	IF TON_2.Q THEN(* PrintOk:=TRUE;	*) step:=0;END_IF

END_CASE
END_PROGRAM

(* POU DataLog/ProductionData_Report, ST *)
PROGRAM ProductionData_Report
VAR

	TON_Indo1: TON;
	TON_Indo2: TON;
	TON_Indo3: TON;
	TON_Indo4: TON;
	TON_Newdaydly: TON;
	TON_NEWDAY: TON;
	TON_NewdaydlyError: TON;
	TON_writedly: TON;
	TON_Opendly: TON;
END_VAR
	ProductionData_ReportData1.SERIALNO	:=DINT_TO_STRING(SerialNo);
		ProductionData_ReportData1.SDATE	:=(wTodayToHmiFinal);
		ProductionData_ReportData1.BAGNO	:=DINT_TO_STRING(CARTONNO_DIS);
		ProductionData_ReportData1.COUNTCODE	:=(COUNT_DIS);
		ProductionData_ReportData1.LOTNO	:=(LOTNO_DIS);
		ProductionData_ReportData1.DFLTNETWEIGHT	:=(Default_NetWeight_Report);
		ProductionData_ReportData1.ACTNETWEIGHT	:=(Actual_NetWeight_Report);



FB_FileOpen_Indo(
	sNetId:='192.168.225.76.1.1',
	sPathName:= ReportPath_Final_2,
	nMode:=FOPEN_MODEAPPEND ,
	ePath:=PATH_GENERIC ,
	bExecute:= ,
	tTimeout:=T#2s ,
	bBusy=> ,
	bError=> ,
	nErrId=> ,
	hFile=> );

FB_FileWrite_Indo(
	sNetId:='192.168.225.76.1.1',
	hFile:=FB_FileOpen_Indo.hFile ,
	pWriteBuff:=ADR(ProductionDataValues_IndoPrint_Com),
	cbWriteLen:=LEN(ProductionDataValues_IndoPrint_Com),
	bExecute:= ,
	tTimeout:=T#2s ,
	bBusy=> ,
	bError=> ,
	nErrId=> ,
	cbWrite=> );


FB_FileClose_Indo(
	sNetId:='192.168.225.76.1.1',
	hFile:=FB_FileOpen_Indo.hFile ,
	bExecute:= ,
	tTimeout:=T#2s ,
	bBusy=> ,
	bError=> ,
	nErrId=> );

FB_FileDelete_Indo(
	sNetId:='192.168.225.76.1.1',
	sPathName:= ReportPath_Final_2,
	ePath:=PATH_GENERIC ,
	bExecute:= ,
	tTimeout:=T#2s ,
	bBusy=> ,
	bError=> ,
	nErrId=> );

R_TRIG_IndoPrint(CLK:=( bANewDay OR testbit)  , Q=> );

CASE IndoReport OF
0:	  IF TON_NEWDAY.Q   THEN	sOldDay := sDay;TON_Newdaydly(IN:=TRUE , PT:=t#0.2s , Q=> , ET=> );
		IF TON_Newdaydly.Q THEN
		bANewDay:=FALSE;IndoReport:=1; SerialNo:=1;FB_FileOpen_Indo.bExecute:=TRUE;END_IF END_IF

1:	TON_Newdaydly(IN:=FALSE);TON_NEWDAY(IN:=FALSE);
	IF NOT FB_FileOpen_Indo.bBusy AND NOT FB_FileOpen_Indo.bError AND FB_FileOpen_Indo.hFile>0 THEN ReportHead1_Indo:=TRUE;END_IF

	IF ReportHead1_Indo THEN
	ProductionData_IndoPrint:= CONCAT( 'SL NO',',');
	ProductionData_IndoPrint:=	 CONCAT( ProductionData_IndoPrint,'DATE/TIME');
		ProductionData_IndoPrint:= CONCAT( ProductionData_IndoPrint,',');
	ProductionData_IndoPrint:=	 CONCAT( ProductionData_IndoPrint,'BAG NO');
		ProductionData_IndoPrint:= CONCAT( ProductionData_IndoPrint,',');
	ProductionData_IndoPrint:=	 CONCAT( ProductionData_IndoPrint,'COUNT');
		ProductionData_IndoPrint:=CONCAT( ProductionData_IndoPrint,',');
	ProductionData_IndoPrint:=	 CONCAT( ProductionData_IndoPrint,'LOT NO');
		ProductionData_IndoPrint:=CONCAT( ProductionData_IndoPrint,',');
	ProductionData_IndoPrint:=	 CONCAT( ProductionData_IndoPrint,'DFLT NET WT');
		ProductionData_IndoPrint:=CONCAT( ProductionData_IndoPrint,',');
	ProductionData_IndoPrint:=	 CONCAT( ProductionData_IndoPrint,'ACT NET WT');
		ProductionData_IndoPrint:= CONCAT( ProductionData_IndoPrint,'$0A');
	IndoReport:=7; END_IF

2:	PROCESSCOMPLETE:=FALSE;ReportHead1_Indo:=FALSE;ProductionDataValues_IndoPrint_Com:=ProductionData_IndoPrint;
	TON_Indo1(IN:=TRUE , PT:=t#5s , Q=> , ET=> );
	FB_FileWrite_Indo.bExecute:=TRUE;
	IF NOT FB_FileWrite_Indo.bBusy AND NOT FB_FileWrite_Indo.bError AND FB_FileWrite_Indo.hFile>0 AND TON_Indo1.Q THEN IndoReport:=IndoReport+1; END_IF

3:	ProductionDataValues_IndoPrint_Com:=ProductionData_IndoPrint;
	FB_FileWrite_Indo.bExecute:=TRUE;
	IF NOT FB_FileWrite_Indo.bBusy AND NOT FB_FileWrite_Indo.bError THEN IndoReport:=IndoReport+1; END_IF

4:	FB_FileWrite_Indo.bExecute:=FALSE;ProductionData_IndoPrint:='';IndoReport:=IndoReport+1;

5:	ReportHead2_Indo:=TRUE;
	IF ReportHead2_Indo THEN IndoReport:=IndoReport+1;END_IF

6:	ProductionData_IndoPrint:=	 CONCAT( ProductionData_IndoPrint,'Cn13Wt');
		ProductionData_IndoPrint:=CONCAT( ProductionData_IndoPrint,',');
	ProductionData_IndoPrint:=	 CONCAT( ProductionData_IndoPrint,'Cn14Wt');
		ProductionData_IndoPrint:=CONCAT( ProductionData_IndoPrint,',');
	ProductionData_IndoPrint:=	 CONCAT( ProductionData_IndoPrint,'Cn15Wt');
		ProductionData_IndoPrint:=CONCAT( ProductionData_IndoPrint,',');
	ProductionData_IndoPrint:=	 CONCAT( ProductionData_IndoPrint,'Cn16Wt');
		ProductionData_IndoPrint:=CONCAT( ProductionData_IndoPrint,',');
	ProductionData_IndoPrint:=	 CONCAT( ProductionData_IndoPrint,'Cn17Wt');
		ProductionData_IndoPrint:=CONCAT( ProductionData_IndoPrint,',');
	ProductionData_IndoPrint:=	 CONCAT( ProductionData_IndoPrint,'Cn18Wt');
		ProductionData_IndoPrint:=CONCAT( ProductionData_IndoPrint,',');
	ProductionData_IndoPrint:=	 CONCAT( ProductionData_IndoPrint,'Cn19Wt');
		ProductionData_IndoPrint:=CONCAT( ProductionData_IndoPrint,',');
	ProductionData_IndoPrint:=	 CONCAT( ProductionData_IndoPrint,'Cn20Wt');
		ProductionData_IndoPrint:=CONCAT( ProductionData_IndoPrint,',');
	ProductionData_IndoPrint:=	 CONCAT( ProductionData_IndoPrint,'Cn21Wt');
		ProductionData_IndoPrint:=CONCAT( ProductionData_IndoPrint,',');
	ProductionData_IndoPrint:=	 CONCAT( ProductionData_IndoPrint,'Cn22Wt');
		ProductionData_IndoPrint:=CONCAT( ProductionData_IndoPrint,',');
	ProductionData_IndoPrint:=	 CONCAT( ProductionData_IndoPrint,'Cn23Wt');
		ProductionData_IndoPrint:=CONCAT( ProductionData_IndoPrint,',');
	ProductionData_IndoPrint:=	 CONCAT( ProductionData_IndoPrint,'Cn24Wt');
		ProductionData_IndoPrint:= CONCAT( ProductionData_IndoPrint,'$0A');
	ReportHead2_Indo:=FALSE;
	IndoReport:=IndoReport+1;

7:	ReportHead1_Indo:=FALSE;ProductionDataValues_IndoPrint_Com:=ProductionData_IndoPrint;
	TON_Indo2(IN:=TRUE , PT:=t#5s , Q=> , ET=> );
	FB_FileWrite_Indo.bExecute:=TRUE;
	IF NOT FB_FileWrite_Indo.bBusy AND NOT FB_FileWrite_Indo.bError  AND TON_Indo2.Q THEN  IndoReport:=IndoReport+1; END_IF

8:	FB_FileWrite_Indo.bExecute:=FALSE;
	FB_FileClose_Indo.bExecute:=TRUE;
	 IF NOT FB_FileClose_Indo.bBusy AND NOT FB_FileClose_Indo.bError THEN FB_FileOpen_Indo.bExecute:=FALSE; IndoReport:=IndoReport+1;END_IF(*ProductionData_IndoPrint:='';*)

9:	FB_FileClose_Indo.bExecute:=FALSE;
	IF ReportSave OR testbit THEN

	FB_FileOpen_Indo.bExecute:=TRUE;
	IF NOT FB_FileOpen_Indo.bBusy AND NOT FB_FileOpen_Indo.bError AND FB_FileOpen_Indo.hFile>0 THEN
	ReportBot1_Indo:=TRUE;END_IF

	IF ReportBot1_Indo THEN IndoReport:=IndoReport+1;END_IF END_IF

10:
	ProductionData_IndoPrint2:= CONCAT(ProductionData_ReportData1.SERIALNO,',');
	ProductionData_IndoPrint2:=	 CONCAT( ProductionData_IndoPrint2,ProductionData_ReportData1.SDATE	);
		ProductionData_IndoPrint2:= CONCAT( ProductionData_IndoPrint2,',');
	ProductionData_IndoPrint2:=	 CONCAT( ProductionData_IndoPrint2,ProductionData_ReportData1.BAGNO	);
		ProductionData_IndoPrint2:= CONCAT( ProductionData_IndoPrint2,',');
	ProductionData_IndoPrint2:=	 CONCAT( ProductionData_IndoPrint2,ProductionData_ReportData1.COUNTCODE);
		ProductionData_IndoPrint2:= CONCAT( ProductionData_IndoPrint2,',');
	ProductionData_IndoPrint2:=	 CONCAT( ProductionData_IndoPrint2,ProductionData_ReportData1.LOTNO);
		ProductionData_IndoPrint2:= CONCAT( ProductionData_IndoPrint2,',');
	ProductionData_IndoPrint2:=	 CONCAT( ProductionData_IndoPrint2,ProductionData_ReportData1.DFLTNETWEIGHT);
		ProductionData_IndoPrint2:= CONCAT( ProductionData_IndoPrint2,',');
	ProductionData_IndoPrint2:=	 CONCAT( ProductionData_IndoPrint2,ProductionData_ReportData1.ACTNETWEIGHT);
		ProductionData_IndoPrint2:= CONCAT( ProductionData_IndoPrint2,'$0A');
	ReportBot1_Indo:=FALSE;ReportSave:=FALSE;
	IndoReport:=15;


11:	ProductionDataValues_IndoPrint_Com:=ProductionData_IndoPrint2;
	TON_Indo3(IN:=TRUE , PT:=t#5s , Q=> , ET=> );
	FB_FileWrite_Indo.bExecute:=TRUE;
	IF NOT FB_FileWrite_Indo.bBusy AND NOT FB_FileWrite_Indo.bError AND TON_Indo3.Q THEN
	 IndoReport:=IndoReport+1; END_IF

12:	FB_FileWrite_Indo.bExecute:=FALSE;IndoReport:=IndoReport+1;

13:	ReportBot2_Indo:=TRUE;
	IF ReportBot2_Indo THEN IndoReport:=IndoReport+1;END_IF

14:	ReportBot2_Indo:=FALSE;
	IndoReport:=IndoReport+1;

15:	ProductionDataValues_IndoPrint_Com:=ProductionData_IndoPrint2;
	TON_Indo4(IN:=TRUE , PT:=t#5s , Q=> , ET=> );
	FB_FileWrite_Indo.bExecute:=TRUE; IndoReport:=IndoReport+1;


16:	IF NOT FB_FileWrite_Indo.bBusy AND NOT FB_FileWrite_Indo.bError THEN
	FB_FileWrite_Indo.bExecute:=FALSE; IndoReport:=IndoReport+1;END_IF


17:	TON_Indo3(IN:=FALSE);TON_Indo4(IN:=FALSE);TON_Indo2(IN:=FALSE);
	TON_Indo1(IN:=FALSE);FB_FileWrite_Indo.bExecute:=FALSE;IndoReport:=IndoReport+1;

